		// Axis not coupled	
		IF NOT _stAXIS_REF.Status.Coupled THEN
			FB_MC2_AxisBasic_M_nMC_SetPositionRelative_iState:= 001;
		ELSE
			FB_MC2_AxisBasic_M_nMC_SetPositionRelative_iState:= 010;
		END_IF
	END_IF
ELSE
	FB_MC2_AxisBasic_M_nMC_SetPositionRelative_fbExecute_R_TRIG(CLK:= FALSE);
	FB_MC2_AxisBasic_M_nMC_SetPositionRelative_iState:= 000;
	IF FB_MC2_AxisBasic_M_nMC_SetPositionRelative_bExecute THEN
		M_nMC_SetPositionRelative:= Tc3_HBI_System.cMAPPING_ERROR;
	END_IF
	RETURN;
END_IF


//**********************************
// Main sequence
//**********************************
CASE FB_MC2_AxisBasic_M_nMC_SetPositionRelative_iState OF

	000: 	// Do nothing
	
	001:	// Set Axis position
			M_nMC_SetPositionRelative:= Tc3_HBI_System.cRUNNING;
			IF _stAXIS_REF.NcToPlc.AxisID > 0 THEN
				FB_MC2_AxisBasic_M_nMC_SetPositionRelative_fbMC2_SetPosition(Axis:= _stAXIS_REF, Execute:= FALSE); 
				FB_MC2_AxisBasic_M_nMC_SetPositionRelative_fbMC2_SetPosition(Axis:= _stAXIS_REF, Execute:= TRUE, Position:= FB_MC2_AxisBasic_M_nMC_SetPositionRelative_lrPosition); 
				FB_MC2_AxisBasic_M_nMC_SetPositionRelative_iState:= FB_MC2_AxisBasic_M_nMC_SetPositionRelative_iState +1;
			END_IF
			
	002:	// Set Axis position - Done
			M_nMC_SetPositionRelative:= Tc3_HBI_System.cRUNNING;
			FB_MC2_AxisBasic_M_nMC_SetPositionRelative_fbMC2_SetPosition(Axis:= _stAXIS_REF, Execute:= TRUE); 
			
			// Error handling
			IF FB_MC2_AxisBasic_M_nMC_SetPositionRelative_fbMC2_SetPosition.Error THEN
				M_nError(FB_MC2_AxisBasic_M_nMC_SetPositionRelative_fbMC2_SetPosition.ErrorID);
				M_nMC_SetPositionRelative:= FB_MC2_AxisBasic_M_nMC_SetPositionRelative_fbMC2_SetPosition.ErrorID;
			ELSE
				// Done
				IF FB_MC2_AxisBasic_M_nMC_SetPositionRelative_fbMC2_SetPosition.Done THEN
					FB_MC2_AxisBasic_M_nMC_SetPositionRelative_fbMC2_SetPosition(Axis:= _stAXIS_REF, Execute:= FALSE); 
					FB_MC2_AxisBasic_M_nMC_SetPositionRelative_iState:= 020;
				END_IF
			END_IF
		
	010:	// Coupled
			M_nMC_SetPositionRelative:= Tc3_HBI_System.cCOUPLED;
			IF NOT FB_MC2_AxisBasic_M_nMC_SetPositionRelative_bExecute THEN
				FB_MC2_AxisBasic_M_nMC_SetPositionRelative_fbMC2_SetPosition(Axis:= _stAXIS_REF, Execute:= FALSE); 
				FB_MC2_AxisBasic_M_nMC_SetPositionRelative_iState:= 000;
			END_IF	

	020:	// Done
			M_nMC_SetPositionRelative:= Tc3_HBI_System.cCOMPLETE;
			
			IF NOT FB_MC2_AxisBasic_M_nMC_SetPositionRelative_bExecute THEN
				FB_MC2_AxisBasic_M_nMC_SetPositionRelative_fbMC2_SetPosition(Axis:= _stAXIS_REF, Execute:= FALSE); 
				FB_MC2_AxisBasic_M_nMC_SetPositionRelative_iState:= 000;
			END_IF	
		
ELSE
	FB_MC2_AxisBasic_M_nMC_SetPositionRelative_iState:= 000;
END_CASE
END_METHOD

//	The result of the method is an unsigned double integer
//	0 = idle 
//	1 = coupled
//	2 = starting
//	3 = running
//	4 = aborted
// 	5 = no hardware connected
// 	6 = Spare
//	7 = pointer or index error
//	8 = mapping error
//	9 = parameter error
//	10 = complete
//	Any other number = ErrorID
METHOD PUBLIC M_nMC_SetScaleFactor : UDINT
VAR_INPUT
	bExecute: BOOL;
	lrScaleFactor: LREAL;
END_VAR
// Local variable
FB_MC2_AxisBasic_M_nMC_SetScaleFactor_bExecute:= bExecute;
FB_MC2_AxisBasic_M_nMC_SetScaleFactor_lrScaleFactor:= lrScaleFactor;

//**********************************
// Reset 
//**********************************
IF _bReset THEN
	IF _bError THEN
		FB_MC2_AxisBasic_M_nMC_SetScaleFactor_fbMC2_SetEncoderScalingFactor(Axis:= _stAXIS_REF, Execute:= FALSE);
		FB_MC2_AxisBasic_M_nMC_SetScaleFactor_iState:= 000;
	END_IF	
END_IF

//**********************************
// Wait for execute
//**********************************
IF _stAXIS_REF.NcToPlc.AxisID > 0 THEN
	FB_MC2_AxisBasic_M_nMC_SetScaleFactor_fbExecute_R_TRIG(CLK:= FB_MC2_AxisBasic_M_nMC_SetScaleFactor_bExecute);
	IF FB_MC2_AxisBasic_M_nMC_SetScaleFactor_fbExecute_R_TRIG.Q THEN
		FB_MC2_AxisBasic_M_nMC_SetScaleFactor_fbMC2_SetEncoderScalingFactor(Axis:= _stAXIS_REF, Execute:= FALSE, ScalingFactor:= FB_MC2_AxisBasic_M_nMC_SetScaleFactor_lrScaleFactor, Mode:= ENCODERSCALINGMODE_RELATIVE);
		
		// Axis not coupled	
		IF NOT _stAXIS_REF.Status.Coupled THEN
			FB_MC2_AxisBasic_M_nMC_SetScaleFactor_iState:= 001;
		ELSE
			FB_MC2_AxisBasic_M_nMC_SetScaleFactor_iState:= 010;
		END_IF
	END_IF
ELSE
	FB_MC2_AxisBasic_M_nMC_SetScaleFactor_fbExecute_R_TRIG(CLK:= FALSE);
	FB_MC2_AxisBasic_M_nMC_SetScaleFactor_iState:= 000;
	IF FB_MC2_AxisBasic_M_nMC_SetScaleFactor_bExecute THEN
		M_nMC_SetScaleFactor:= Tc3_HBI_System.cMAPPING_ERROR;
	END_IF
	RETURN;
END_IF

//**********************************
// Parameter check 
//**********************************
IF FB_MC2_AxisBasic_M_nMC_SetScaleFactor_bExecute THEN
	IF FB_MC2_AxisBasic_M_nMC_SetScaleFactor_lrScaleFactor = 0.0 THEN
		M_nMC_SetScaleFactor:= Tc3_HBI_System.cPARAMETER_ERROR;
		RETURN;
	END_IF
END_IF


//**********************************
// Main sequence
//**********************************
CASE FB_MC2_AxisBasic_M_nMC_SetScaleFactor_iState OF

	000: 	// Do nothing
	
	001:	// Check parameter input
			M_nMC_SetScaleFactor:= Tc3_HBI_System.cSTARTING;
			IF _stAXIS_REF.NcToPlc.AxisID > 0 THEN
				IF FB_MC2_AxisBasic_M_nMC_SetScaleFactor_lrScaleFactor > 0.0 THEN 
					FB_MC2_AxisBasic_M_nMC_SetScaleFactor_iState:= 2;
				ELSE
					M_nMC_SetScaleFactor:= Tc3_HBI_System.cPARAMETER_ERROR;
					IF NOT FB_MC2_AxisBasic_M_nMC_SetScaleFactor_bExecute THEN
						FB_MC2_AxisBasic_M_nMC_SetScaleFactor_iState:= 000;
					END_IF
				END_IF
			END_IF

	002:	// Set axis scale factor
			M_nMC_SetScaleFactor:= Tc3_HBI_System.cRUNNING;
			FB_MC2_AxisBasic_M_nMC_SetScaleFactor_fbMC2_SetEncoderScalingFactor(Axis:= _stAXIS_REF, Execute:= TRUE, ScalingFactor:= FB_MC2_AxisBasic_M_nMC_SetScaleFactor_lrScaleFactor, Mode:= ENCODERSCALINGMODE_RELATIVE);
			
			// Error handling
			IF FB_MC2_AxisBasic_M_nMC_SetScaleFactor_fbMC2_SetEncoderScalingFactor.Error THEN
				M_nError(FB_MC2_AxisBasic_M_nMC_SetScaleFactor_fbMC2_SetEncoderScalingFactor.ErrorID);
				M_nMC_SetScaleFactor:= FB_MC2_AxisBasic_M_nMC_SetScaleFactor_fbMC2_SetEncoderScalingFactor.ErrorID;
			ELSE
				// Done
				IF FB_MC2_AxisBasic_M_nMC_SetScaleFactor_fbMC2_SetEncoderScalingFactor.Done THEN
					FB_MC2_AxisBasic_M_nMC_SetScaleFactor_fbMC2_SetEncoderScalingFactor(Axis:= _stAXIS_REF, Execute:= FALSE);
					FB_MC2_AxisBasic_M_nMC_SetScaleFactor_iState:= 020;
				END_IF
			END_IF
		
	010:	// Coupled
			M_nMC_SetScaleFactor:= Tc3_HBI_System.cCOUPLED;
			IF NOT FB_MC2_AxisBasic_M_nMC_SetScaleFactor_bExecute THEN
				FB_MC2_AxisBasic_M_nMC_SetScaleFactor_fbMC2_SetEncoderScalingFactor(Axis:= _stAXIS_REF, Execute:= FALSE);
				FB_MC2_AxisBasic_M_nMC_SetScaleFactor_iState:= 000;
			END_IF	

	020:	// Done
			M_nMC_SetScaleFactor:= Tc3_HBI_System.cCOMPLETE;

			IF NOT FB_MC2_AxisBasic_M_nMC_SetScaleFactor_bExecute THEN
				FB_MC2_AxisBasic_M_nMC_SetScaleFactor_fbMC2_SetEncoderScalingFactor(Axis:= _stAXIS_REF, Execute:= FALSE);
				FB_MC2_AxisBasic_M_nMC_SetScaleFactor_iState:= 000;
			END_IF	

ELSE
	FB_MC2_AxisBasic_M_nMC_SetScaleFactor_iState:= 000;
END_CASE
END_METHOD

//	The result of the method is an unsigned double integer
//	0 = idle 
//	1 = coupled
//	2 = starting
//	3 = running
//	4 = aborted
// 	5 = no hardware connected
// 	6 = Spare
//	7 = pointer or index error
//	8 = mapping error
//	9 = parameter error
//	10 = complete
//	Any other number = ErrorID
METHOD PUBLIC M_nMC_SetVeloKvFactor : UDINT
VAR_INPUT
	bExecute: BOOL;
	lrKvFactor: LREAL;
END_VAR
// Local variable
FB_MC2_AxisBasic_M_nMC_SetVeloKvFactor_bExecute:= bExecute;
FB_MC2_AxisBasic_M_nMC_SetVeloKvFactor_lrKvFactor:= lrKvFactor;

//**********************************
// Reset 
//**********************************
IF _bReset THEN
	IF _bError THEN
		FB_MC2_AxisBasic_M_nMC_SetVeloKvFactor_fbADSWRITE(WRITE:= FALSE); 
		FB_MC2_AxisBasic_M_nMC_SetVeloKvFactor_iState:= 000;
	END_IF
END_IF

//**********************************
// Parameter check 
//**********************************
IF FB_MC2_AxisBasic_M_nMC_SetVeloKvFactor_bExecute THEN
	IF FB_MC2_AxisBasic_M_nMC_SetVeloKvFactor_lrKvFactor <= 0.0 THEN
		M_nMC_SetVeloKvFactor:= Tc3_HBI_System.cPARAMETER_ERROR;
		RETURN;
	END_IF	
END_IF


//**********************************
// Wait for execute
//**********************************
IF _stAXIS_REF.NcToPlc.AxisID > 0 THEN
	FB_MC2_AxisBasic_M_nMC_SetVeloKvFactor_fbExecute_R_TRIG(CLK:= FB_MC2_AxisBasic_M_nMC_SetVeloKvFactor_bExecute);
	IF FB_MC2_AxisBasic_M_nMC_SetVeloKvFactor_fbExecute_R_TRIG.Q THEN
		FB_MC2_AxisBasic_M_nMC_SetVeloKvFactor_iState:= 001;
	END_IF
ELSE
	FB_MC2_AxisBasic_M_nMC_SetVeloKvFactor_fbExecute_R_TRIG(CLK:= FALSE);
	FB_MC2_AxisBasic_M_nMC_SetVeloKvFactor_iState:= 000;
	IF FB_MC2_AxisBasic_M_nMC_SetVeloKvFactor_bExecute THEN
		M_nMC_SetVeloKvFactor:= Tc3_HBI_System.cMAPPING_ERROR;
	END_IF
	RETURN;
END_IF


//**********************************
// Main sequence
//**********************************
CASE FB_MC2_AxisBasic_M_nMC_SetVeloKvFactor_iState OF

	000: 	// Do nothing

	001:	// Set Velo Kv faktor
			IF FB_MC2_AxisBasic_M_nMC_SetVeloKvFactor_bExecute THEN				
				M_nMC_SetVeloKvFactor:= Tc3_HBI_System.cSTARTING;
				FB_MC2_AxisBasic_M_nMC_SetVeloKvFactor_fbADSWRITE(WRITE:= FALSE);
				FB_MC2_AxisBasic_M_nMC_SetVeloKvFactor_fbADSWRITE(
					NETID:= '', 
					PORT:= 501, 
					IDXGRP:= 16#6000 + _stAXIS_REF.NcToPlc.AxisId, 
					IDXOFFS:= 16#102, 
					LEN:= SIZEOF(FB_MC2_AxisBasic_M_nMC_SetVeloKvFactor_lrKvFactor), 
					SRCADDR:= ADR(FB_MC2_AxisBasic_M_nMC_SetVeloKvFactor_lrKvFactor), 
					WRITE:= TRUE, 
					TMOUT:= Tc2_System.DEFAULT_ADS_TIMEOUT, 
					BUSY=> , 
					ERR=> , 
					ERRID=> );
	 
				FB_MC2_AxisBasic_M_nMC_SetVeloKvFactor_iState:= FB_MC2_AxisBasic_M_nMC_SetVeloKvFactor_iState +1;
			ELSE
				FB_MC2_AxisBasic_M_nMC_SetVeloKvFactor_iState:= 000;
			END_IF	
	
	002:	// Done	
			M_nMC_SetVeloKvFactor:= Tc3_HBI_System.cRUNNING;	
			FB_MC2_AxisBasic_M_nMC_SetVeloKvFactor_fbADSWRITE(WRITE:= TRUE);
		
			// Error handling
			IF FB_MC2_AxisBasic_M_nMC_SetVeloKvFactor_fbADSWRITE.ERR THEN
				M_nError(nErrorID:= FB_MC2_AxisBasic_M_nMC_SetVeloKvFactor_fbADSWRITE.ERRID);
				M_nMC_SetVeloKvFactor:= FB_MC2_AxisBasic_M_nMC_SetVeloKvFactor_fbADSWRITE.ERRID;
			ELSE
				// Done
				IF NOT FB_MC2_AxisBasic_M_nMC_SetVeloKvFactor_fbADSWRITE.BUSY THEN
					FB_MC2_AxisBasic_M_nMC_SetVeloKvFactor_fbADSWRITE(WRITE:= FALSE); 
					FB_MC2_AxisBasic_M_nMC_SetVeloKvFactor_iState:= FB_MC2_AxisBasic_M_nMC_SetVeloKvFactor_iState +1;
				END_IF
			END_IF
			
	003:	// Done
			M_nMC_SetVeloKvFactor:= Tc3_HBI_System.cCOMPLETE;
			
			IF NOT FB_MC2_AxisBasic_M_nMC_SetVeloKvFactor_bExecute THEN	
				FB_MC2_AxisBasic_M_nMC_SetVeloKvFactor_iState:= 000;
			END_IF	
		
ELSE
	FB_MC2_AxisBasic_M_nMC_SetVeloKvFactor_iState:= 000;
END_CASE
END_METHOD

//	The result of the method is an unsigned double integer
//	0 = idle 
//	1 = coupled
//	2 = starting
//	3 = running
//	4 = aborted
// 	5 = no hardware connected
// 	6 = Spare
//	7 = pointer or index error
//	8 = mapping error
//	9 = parameter error
//	10 = complete
//	Any other number = ErrorID
METHOD PUBLIC M_nReset : UDINT
VAR_INPUT
	bExecute: BOOL;
END_VAR
// Local variable
FB_MC2_AxisBasic_M_nReset_bExecute:= bExecute;

//**********************************
// Wait for execute
//**********************************
FB_MC2_AxisBasic_M_nReset_fbExecute_R_TRIG(CLK:= FB_MC2_AxisBasic_M_nReset_bExecute);
IF FB_MC2_AxisBasic_M_nReset_fbExecute_R_TRIG.Q THEN
	FB_MC2_AxisBasic_M_nReset_fbMC2_Reset(Axis:= _stAXIS_REF, Execute:= FALSE);
	SUPER^.M_nReset(bExecute:= FALSE);
	FB_MC2_AxisBasic_M_nReset_bError:= _bError;
	FB_MC2_AxisBasic_M_nReset_iState:= 001;
END_IF	


//**********************************
// Main sequence
//**********************************
CASE FB_MC2_AxisBasic_M_nReset_iState OF

	000: 	// Do nothing
		
	001:	// Reset father	
			M_nReset:= Tc3_HBI_System.cRUNNING;
			FB_MC2_AxisBasic_M_nReset_nStatus:= SUPER^.M_nReset(bExecute:= TRUE);
			
			// Error handling
			IF FB_MC2_AxisBasic_M_nReset_nStatus > Tc3_HBI_System.cCOMPLETE THEN
				SUPER^.M_nReset(bExecute:= FALSE);		
				IF _stAXIS_REF.Status.Coupled THEN
					FB_MC2_AxisBasic_M_nReset_iState:= 020;
				ELSE
					FB_MC2_AxisBasic_M_nReset_iState:= 030;
				END_IF
			END_IF

			// Done
			IF FB_MC2_AxisBasic_M_nReset_nStatus = Tc3_HBI_System.cCOUPLED OR FB_MC2_AxisBasic_M_nReset_nStatus = Tc3_HBI_System.cCOMPLETE THEN
				SUPER^.M_nReset(bExecute:= FALSE);		
				IF _stAXIS_REF.Status.Coupled THEN
					FB_MC2_AxisBasic_M_nReset_iState:= 020;
				ELSE
					FB_MC2_AxisBasic_M_nReset_iState:= 030;
				END_IF
			END_IF
			
	020:	// Coupled
			M_nReset:= Tc3_HBI_System.cCOUPLED;
			IF NOT FB_MC2_AxisBasic_M_nReset_bExecute THEN
				FB_MC2_AxisBasic_M_nReset_fbMC2_Reset(Axis:= _stAXIS_REF, Execute:= FALSE);
				SUPER^.M_nReset(bExecute:= FALSE);		
				FB_MC2_AxisBasic_M_nReset_iState:= 000;
			END_IF	
	
	030:	// Done
			M_nReset:= Tc3_HBI_System.cCOMPLETE;
			IF NOT FB_MC2_AxisBasic_M_nReset_bExecute THEN
				FB_MC2_AxisBasic_M_nReset_fbMC2_Reset(Axis:= _stAXIS_REF, Execute:= FALSE);
				SUPER^.M_nReset(bExecute:= FALSE);		
				FB_MC2_AxisBasic_M_nReset_iState:= 000;
			END_IF

ELSE
	FB_MC2_AxisBasic_M_nReset_iState:= 000;
END_CASE
END_METHOD

PROPERTY PUBLIC P_bAdvancedSlaveDynamics : BOOL
SET
FB_MC2_AxisBasic_M_nMC_GearInMultiMaster_bAdvancedSlaveDynamics:= P_bAdvancedSlaveDynamics;
END_SET
END_PROPERTY

PROPERTY PUBLIC P_bInGear : BOOL
GET
P_bInGear:= _stAXIS_REF.Status.Coupled;
END_GET
END_PROPERTY

PROPERTY PUBLIC P_lrAbsolutePhaseShift  : lreal
GET
P_lrAbsolutePhaseShift:= FB_MC2_AxisBasic_M_nMC_PhasingAbsolute_lrAbsolutePhaseShift;
END_GET
END_PROPERTY

PROPERTY PUBLIC P_lrCoveredPhaseShift : lreal
GET
P_lrCoveredPhaseShift:= FB_MC2_AxisBasic_M_nMC_PhasingRelative_lrCoveredPhaseShift;
END_GET
END_PROPERTY

PROPERTY PUBLIC P_lrGearRatio1 : LREAL
SET
FB_MC2_AxisBasic_M_nMC_GearInMultiMaster_lrGearRatio1:= P_lrGearRatio1;
END_SET
END_PROPERTY

PROPERTY PUBLIC P_lrGearRatio2 : LREAL
SET
FB_MC2_AxisBasic_M_nMC_GearInMultiMaster_lrGearRatio2:= P_lrGearRatio2;
END_SET
END_PROPERTY

PROPERTY PUBLIC P_lrGearRatio3 : LREAL
SET
FB_MC2_AxisBasic_M_nMC_GearInMultiMaster_lrGearRatio3:= P_lrGearRatio3;
END_SET
END_PROPERTY

PROPERTY PUBLIC P_lrGearRatio4 : LREAL
SET
FB_MC2_AxisBasic_M_nMC_GearInMultiMaster_lrGearRatio4:= P_lrGearRatio4;
END_SET
END_PROPERTY

PROPERTY PUBLIC P_lrMaxVelocity : LREAL
GET
P_lrMaxVelocity:= FB_MC2_AxisBasic_M_nMC_ReadParameter_lrMaxVelocity;
END_GET
END_PROPERTY

PROPERTY PUBLIC P_lrModuloFactor : LREAL
GET
IF FB_MC2_AxisBasic_M_nMC_SetModuloFactor_lrModuloFactor = 0 THEN
	FB_MC2_AxisBasic_M_nMC_SetModuloFactor_lrModuloFactor:= 360.0;
	P_lrModuloFactor:= FB_MC2_AxisBasic_M_nMC_SetModuloFactor_lrModuloFactor;
ELSE
	P_lrModuloFactor:= FB_MC2_AxisBasic_M_nMC_SetModuloFactor_lrModuloFactor;
END_IF
END_GET
END_PROPERTY

END_FUNCTION_BLOCK

// MOTION/POUs/FBs/Compact/FB_MC2_Compact
//------------------------------------------------------------------------------------------
//                                                                                        	
//***************************** Beckhoff TwinCAT Examples **********************************
//                                                                                        	
//************************************* WARNING ********************************************
// This program is only an example. If it is used as a control program in any real        	
// application, Beckhoff is not responsible for any malfunction, loss or damage           	
// which could arise by using this program!                                               	
//                                                                                        	
//*************************************  Program Info. *************************************
//                                                                                        	
// PLC program name:       	FB_MC2_Compact (FB)                                          	
// Hardware platform:      	TwinCat PTP v3.1.4022				                          	                                  	
//                                                                                        	
// ======================================================================================== 
//         Version       Date                        Remarks                              	
// ======================================================================================== 
//         3.1      27 feb 2018                First release of this example  
//         3.7.1.1		 09 may 2018    			 Next release of this example   
// ======================================================================================== 
//                                                                                        	
//******************************* Aims OF this PLC PROGRAM *********************************
//                                                                                        	
// MC2 servo axis compact						 			                                      	
// Add axis error message 																                      	
//                                                                                        	
//----------------------------------------------------------------------------------------- 
FUNCTION_BLOCK FB_MC2_Compact EXTENDS FB_Basic IMPLEMENTS I_MC2_Compact
VAR
//***************************
// Property variables
//***************************
	_stAXIS_REF: Tc2_MC2.AXIS_REF;
	_eBufferMode: MC_BufferMode:= Tc2_MC2.MC_Aborting;
	_bHardwareConnected: BOOL;	
	_stDriveAddress: ST_DriveAddress;
	_stDynamic: _ST_MC2_Dynamic;
	_sMessage: STRING(80);
	
//***************************
// Metods variable
//***************************
	FB_MC2_Compact_M_nMC_Dynamic_bExecute: BOOL;
	FB_MC2_Compact_M_nMC_Dynamic_lrAcceleration: LREAL;
	FB_MC2_Compact_M_nMC_Dynamic_lrDeceleration: LREAL;
	FB_MC2_Compact_M_nMC_Dynamic_lrJerk: LREAL;

	FB_MC2_Compact_M_nMC_Halt_bExecute: BOOL;
	FB_MC2_Compact_M_nMC_Halt_iState: INT;
	FB_MC2_Compact_M_nMC_Halt_fbExecute_R_TRIG: R_TRIG;
	FB_MC2_Compact_M_nMC_Halt_fbMC2_Halt1: Tc2_MC2.MC_Halt;
	FB_MC2_Compact_M_nMC_Halt_fbMC2_Halt2: Tc2_MC2.MC_Halt;

	FB_MC2_Compact_M_nMC_Home_bExecute: BOOL;
	FB_MC2_Compact_M_nMC_Home_lrPosition: LREAL;
	FB_MC2_Compact_M_nMC_Home_bCalibrationCam: BOOL;
	FB_MC2_Compact_M_nMC_Home_eHomingMode: MC_HomingMode;
	FB_MC2_Compact_M_nMC_Home_iState: INT;
	FB_MC2_Compact_M_nMC_Home_fbExecute_R_TRIG: Tc2_Standard.R_TRIG;
	FB_MC2_Compact_M_nMC_Home_fbMC2_Halt: Tc2_MC2.MC_Halt;
	FB_MC2_Compact_M_nMC_Home_fbMC2_Home: Tc2_MC2.MC_Home;
	
	FB_MC2_Compact_M_nMC_HomeReset_bExecute: BOOL;
	FB_MC2_Compact_M_nMC_HomeReset_iState: INT;
	FB_MC2_Compact_M_nMC_HomeReset_fbExecute_R_TRIG: Tc2_Standard.R_TRIG;
	FB_MC2_Compact_M_nMC_HomeReset_fbMC2_Home: Tc2_MC2.MC_Home;

	FB_MC2_Compact_M_nMC_Jog_bForward: BOOL;
	FB_MC2_Compact_M_nMC_Jog_bBackwards: BOOL;
	FB_MC2_Compact_M_nMC_Jog_lrVelocity: LREAL;
	FB_MC2_Compact_M_nMC_Jog_iState: INT;
	FB_MC2_Compact_M_nMC_Jog_fbExecute_R_TRIG1: R_TRIG;
	FB_MC2_Compact_M_nMC_Jog_fbExecute_R_TRIG2: R_TRIG;
	FB_MC2_Compact_M_nMC_Jog_fbMC2_Jog1: Tc2_MC2.MC_Jog;
	FB_MC2_Compact_M_nMC_Jog_fbMC2_Jog2: Tc2_MC2.MC_Jog;

	FB_MC2_Compact_M_nMC_Local_Halt_bExecute: BOOL;
	FB_MC2_Compact_M_nMC_Local_Halt_iState: INT;
	FB_MC2_Compact_M_nMC_Local_Halt_fbExecute_R_TRIG: R_TRIG;
	FB_MC2_Compact_M_nMC_Local_Halt_fbMC2_Halt1: Tc2_MC2.MC_Halt;
	FB_MC2_Compact_M_nMC_Local_Halt_fbMC2_Halt2: Tc2_MC2.MC_Halt;

	FB_MC2_Compact_M_nMC_MoveAbsolute_bExecute: BOOL;
	FB_MC2_Compact_M_nMC_MoveAbsolute_lrPosition: LREAL;
	FB_MC2_Compact_M_nMC_MoveAbsolute_lrVelocity: LREAL;
	FB_MC2_Compact_M_nMC_MoveAbsolute_iState: INT;
	FB_MC2_Compact_M_nMC_MoveAbsolute_fbExecute_R_TRIG: Tc2_Standard.R_TRIG;
	FB_MC2_Compact_M_nMC_MoveAbsolute_fbMC2_MoveAbsolute1: Tc2_MC2.MC_MoveAbsolute;
	FB_MC2_Compact_M_nMC_MoveAbsolute_fbMC2_MoveAbsolute2: Tc2_MC2.MC_MoveAbsolute;

	FB_MC2_Compact_M_nMC_MoveModulo_bExecute: BOOL;
	FB_MC2_Compact_M_nMC_MoveModulo_lrPosition: LREAL;
	FB_MC2_Compact_M_nMC_MoveModulo_lrVelocity: LREAL;
	FB_MC2_Compact_M_nMC_MoveModulo_eDirection: Tc2_MC2.MC_Direction;
	FB_MC2_Compact_M_nMC_MoveModulo_iState: INT;
	FB_MC2_Compact_M_nMC_MoveModulo_fbExecute_R_TRIG: Tc2_Standard.R_TRIG;
	FB_MC2_Compact_M_nMC_MoveModulo_fbMC2_MoveModulo1: Tc2_MC2.MC_MoveModulo;
	FB_MC2_Compact_M_nMC_MoveModulo_fbMC2_MoveModulo2: Tc2_MC2.MC_MoveModulo;

	FB_MC2_Compact_M_nMC_MoveRelative_bExecute: BOOL;
	FB_MC2_Compact_M_nMC_MoveRelative_lrDistance: LREAL;
	FB_MC2_Compact_M_nMC_MoveRelative_lrVelocity: LREAL;
	FB_MC2_Compact_M_nMC_MoveRelative_iState: INT;
	FB_MC2_Compact_M_nMC_MoveRelative_fbExecute_R_TRIG: Tc2_Standard.R_TRIG;
	FB_MC2_Compact_M_nMC_MoveRelative_fbMC2_MoveRelative1: Tc2_MC2.MC_MoveRelative;
	FB_MC2_Compact_M_nMC_MoveRelative_fbMC2_MoveRelative2: Tc2_MC2.MC_MoveRelative;

	FB_MC2_Compact_M_nMC_MoveVelocity_bExecute: BOOL;
	FB_MC2_Compact_M_nMC_MoveVelocity_lrVelocity: LREAL;
	FB_MC2_Compact_M_nMC_MoveVelocity_eDirection: MC_Direction;
	FB_MC2_Compact_M_nMC_MoveVelocity_iState: INT;
	FB_MC2_Compact_M_nMC_MoveVelocity_fbExecute_R_TRIG: Tc2_Standard.R_TRIG;
	FB_MC2_Compact_M_nMC_MoveVelocity_fbMC2_MoveVelocity1: Tc2_MC2.MC_MoveVelocity;
	FB_MC2_Compact_M_nMC_MoveVelocity_fbMC2_MoveVelocity2: Tc2_MC2.MC_MoveVelocity;
	
	FB_MC2_Compact_M_nMC_Power_bEnable: BOOL;
	FB_MC2_Compact_M_nMC_Power_bE_Stop: BOOL;
	FB_MC2_Compact_M_nMC_Power_bE_StopDelay: BOOL;
	FB_MC2_Compact_M_nMC_Power_bEnable_Positive: BOOL;
	FB_MC2_Compact_M_nMC_Power_bEnable_Negative: BOOL;
	FB_MC2_Compact_M_nMC_Power_lrOverride: LREAL := 100.0;
	FB_MC2_Compact_M_nMC_Power_fbStartDelay_TON: Tc2_Standard.TON;
	FB_MC2_Compact_M_nMC_Power_arr_fb_R_TRIG: ARRAY[1..12] OF Tc2_Standard.R_TRIG;
	FB_MC2_Compact_M_nMC_Power_arr_nRet: ARRAY[1..4] OF UDINT;
	FB_MC2_Compact_M_nMC_Power_fbMC2_Power: Tc2_MC2.MC_Power;
	FB_MC2_Compact_M_nMC_Power_fbDelay_TON: Tc2_Standard.TON;
	FB_MC2_Compact_M_nMC_Power_fbPuls_TON: Tc2_Standard.TON;
	FB_MC2_Compact_M_nMC_Power_bReset: BOOL;
	FB_MC2_Compact_M_nMC_Power_iResetState: INT;
	FB_MC2_Compact_M_nMC_Power_bLocal_Halt: BOOL;
	FB_MC2_Compact_M_nMC_Power_bError: BOOL;
	
	FB_MC2_Compact_M_nMC_QuickStop_bExecute: BOOL;
	FB_MC2_Compact_M_nMC_QuickStop_lrDeceleration: LREAL;
	FB_MC2_Compact_M_nMC_QuickStop_lrJerk: LREAL;
	FB_MC2_Compact_M_nMC_QuickStop_bQuickStopRunning: BOOL;
	FB_MC2_Compact_M_nMC_QuickStop_iState: INT;
	FB_MC2_Compact_M_nMC_QuickStop_fbExecute_R_TRIG: Tc2_Standard.R_TRIG;
	FB_MC2_Compact_M_nMC_QuickStop_fbMC2_Stop: Tc2_MC2.MC_Stop;

	FB_MC2_Compact_M_nMC_ReadDriveAddress_bExecute: BOOL;
	FB_MC2_Compact_M_nMC_ReadDriveAddress_iState: INT;
	FB_MC2_Compact_M_nMC_ReadDriveAddress_bError: BOOL;
	FB_MC2_Compact_M_nMC_ReadDriveAddress_fbReadDriveAddress: Tc2_MC2.MC_ReadDriveAddress;

	FB_MC2_Compact_M_nMC_Stop_bExecute: BOOL;
	FB_MC2_Compact_M_nMC_Stop_iState: INT;
	FB_MC2_Compact_M_nMC_Stop_fbExecute_R_TRIG: R_TRIG;
	FB_MC2_Compact_M_nMC_Stop_fbMC2_Stop1: Tc2_MC2.MC_Stop;
	FB_MC2_Compact_M_nMC_Stop_fbMC2_Stop2: Tc2_MC2.MC_Stop;

	FB_MC2_Compact_M_nReset_bExecute: BOOL;
	FB_MC2_Compact_M_nReset_iState: INT;
	FB_MC2_Compact_M_nReset_fbExecute_R_TRIG: Tc2_Standard.R_TRIG;
	FB_MC2_Compact_M_nReset_fbMC2_Reset: Tc2_MC2.MC_Reset;
	FB_MC2_Compact_M_nReset_fbMC2_Stop: Tc2_MC2.MC_Stop;
	FB_MC2_Compact_M_nReset_nStatus: UDINT;
END_VAR

//	The result of the method is an unsigned double integer
//	0 = idle 
//	1 = coupled
//	2 = starting
//	3 = running
//	4 = aborted
// 	5 = no hardware connected
// 	6 = Spare
//	7 = pointer or index error
//	8 = mapping error
//	9 = parameter error
//	10 = complete
//	Any other number = ErrorID
METHOD PUBLIC M_nMC_Dynamic : UDINT
VAR_INPUT
	bExecute: BOOL;
	lrAcceleration: LREAL;
	lrDeceleration: LREAL;
	lrJerk: LREAL;
END_VAR
// Local variable
FB_MC2_Compact_M_nMC_Dynamic_bExecute:= bExecute;
FB_MC2_Compact_M_nMC_Dynamic_lrAcceleration:= lrAcceleration;
FB_MC2_Compact_M_nMC_Dynamic_lrDeceleration:= lrDeceleration;
FB_MC2_Compact_M_nMC_Dynamic_lrJerk:= lrJerk;

//**********************************
// Parameter check 
//**********************************
IF FB_MC2_Compact_M_nMC_Dynamic_bExecute THEN
	IF FB_MC2_Compact_M_nMC_Dynamic_lrAcceleration < 0.0 OR FB_MC2_Compact_M_nMC_Dynamic_lrDeceleration < 0.0 OR FB_MC2_Compact_M_nMC_Dynamic_lrJerk < 0.0 THEN
		M_nMC_Dynamic:= Tc3_HBI_System.cPARAMETER_ERROR;
		RETURN;
	END_IF

	// Check for Axis
	IF _stAXIS_REF.NcToPlc.AxisID = 0 THEN
		RETURN;
	ELSE	
		// Update dynamic
		THIS^._stDynamic.lrAcceleration:= FB_MC2_Compact_M_nMC_Dynamic_lrAcceleration;
		THIS^._stDynamic.lrDeceleration:= FB_MC2_Compact_M_nMC_Dynamic_lrDeceleration;
		THIS^._stDynamic.lrJerk:= FB_MC2_Compact_M_nMC_Dynamic_lrJerk;
		M_nMC_Dynamic:= Tc3_HBI_System.cCOMPLETE;
	END_IF
	
END_IF
END_METHOD

//	The result of the method is an unsigned double integer
//	0 = idle 
//	1 = coupled
//	2 = starting
//	3 = running
//	4 = aborted
// 	5 = no hardware connected
// 	6 = Spare
//	7 = pointer or index error
//	8 = mapping error
//	9 = parameter error
//	10 = complete
//	Any other number = ErrorID
METHOD PUBLIC M_nMC_Halt : UDINT
VAR_INPUT
	bExecute: BOOL;
END_VAR
// Local variable
FB_MC2_Compact_M_nMC_Halt_bExecute:= bExecute;

//**********************************
// Reset 
//**********************************
IF _bReset THEN
	IF _bError THEN
		FB_MC2_Compact_M_nMC_Halt_fbMC2_Halt1(Axis:= _stAXIS_REF, Execute:= FALSE);
		FB_MC2_Compact_M_nMC_Halt_fbMC2_Halt2(Axis:= _stAXIS_REF, Execute:= FALSE);
		FB_MC2_Compact_M_nMC_Halt_iState:= 000;
		_sMessage:= '';
	END_IF
END_IF

//**********************************
// Wait for execute
//**********************************
IF _stAXIS_REF.NcToPlc.AxisID > 0 THEN
	FB_MC2_Compact_M_nMC_Halt_fbExecute_R_TRIG(CLK:= FB_MC2_Compact_M_nMC_Halt_bExecute);
	IF FB_MC2_Compact_M_nMC_Halt_fbExecute_R_TRIG.Q THEN
			FB_MC2_Compact_M_nMC_Halt_fbMC2_Halt1(Axis:= _stAXIS_REF, Deceleration:= _stDynamic.lrDeceleration, Jerk:= _stDynamic.lrJerk, BufferMode:= _eBufferMode);
			FB_MC2_Compact_M_nMC_Halt_fbMC2_Halt2(Axis:= _stAXIS_REF, Deceleration:= _stDynamic.lrDeceleration, Jerk:= _stDynamic.lrJerk, BufferMode:= _eBufferMode);
	
			// Axis not coupled	
			IF NOT _stAXIS_REF.Status.Coupled THEN
				IF FB_MC2_Compact_M_nMC_Halt_fbMC2_Halt1.Execute OR FB_MC2_Compact_M_nMC_Halt_fbMC2_Halt1.Busy THEN
					FB_MC2_Compact_M_nMC_Halt_fbMC2_Halt1(Axis:= _stAXIS_REF, Execute:= FALSE);
					FB_MC2_Compact_M_nMC_Halt_fbMC2_Halt2(Axis:= _stAXIS_REF, Execute:= FALSE);
					FB_MC2_Compact_M_nMC_Halt_fbMC2_Halt2.Execute:= TRUE;
					FB_MC2_Compact_M_nMC_Halt_iState:= 010;
				ELSE
					FB_MC2_Compact_M_nMC_Halt_fbMC2_Halt1(Axis:= _stAXIS_REF, Execute:= FALSE);
					FB_MC2_Compact_M_nMC_Halt_fbMC2_Halt2(Axis:= _stAXIS_REF, Execute:= FALSE);
					FB_MC2_Compact_M_nMC_Halt_fbMC2_Halt1.Execute:= TRUE;
					FB_MC2_Compact_M_nMC_Halt_iState:= 001;
				END_IF
			ELSE
				FB_MC2_Compact_M_nMC_Halt_fbMC2_Halt1(Axis:= _stAXIS_REF, Execute:= FALSE);
				FB_MC2_Compact_M_nMC_Halt_fbMC2_Halt2(Axis:= _stAXIS_REF, Execute:= FALSE);
				FB_MC2_Compact_M_nMC_Halt_iState:= 030;
			END_IF
		
	END_IF
ELSE
	FB_MC2_Compact_M_nMC_Halt_fbExecute_R_TRIG(CLK:= FALSE);
	FB_MC2_Compact_M_nMC_Halt_iState:= 000;
	IF bExecute THEN
		M_nMC_Halt:= Tc3_HBI_System.cMAPPING_ERROR;
	END_IF
	RETURN;
END_IF


//**********************************
// Main sequence
//**********************************
CASE FB_MC2_Compact_M_nMC_Halt_iState OF

	000: 	// Do nothing
	
	001:	// Stop Axis1
			M_nMC_Halt:= Tc3_HBI_System.cSTARTING;
			FB_MC2_Compact_M_nMC_Halt_fbMC2_Halt1(Axis:= _stAXIS_REF);
			FB_MC2_Compact_M_nMC_Halt_fbMC2_Halt2(Axis:= _stAXIS_REF);
		
			// Command aborted
			IF FB_MC2_Compact_M_nMC_Halt_fbMC2_Halt1.CommandAborted THEN
				FB_MC2_Compact_M_nMC_Halt_fbMC2_Halt2.Execute:= FALSE;
				FB_MC2_Compact_M_nMC_Halt_iState:= 040;
			ELSE
				// Error handling
				IF FB_MC2_Compact_M_nMC_Halt_fbMC2_Halt1.Error THEN
					M_nError(FB_MC2_Compact_M_nMC_Halt_fbMC2_Halt1.ErrorID);
					M_nMC_Halt:= FB_MC2_Compact_M_nMC_Halt_fbMC2_Halt1.ErrorID;
					_sMessage:= 'Axis Halt Error';
				ELSE
					// Active
					IF FB_MC2_Compact_M_nMC_Halt_fbMC2_Halt1.Active THEN
						FB_MC2_Compact_M_nMC_Halt_iState:= 002;
					ELSE
						// Done
						IF FB_MC2_Compact_M_nMC_Halt_fbMC2_Halt1.Done THEN
							FB_MC2_Compact_M_nMC_Halt_iState:= 040;
						END_IF
					END_IF	
				END_IF
			END_IF
	
	002:	// Stop Axis
			M_nMC_Halt:= Tc3_HBI_System.cRUNNING;
			FB_MC2_Compact_M_nMC_Halt_fbMC2_Halt1(Axis:= _stAXIS_REF);
			FB_MC2_Compact_M_nMC_Halt_fbMC2_Halt2(Axis:= _stAXIS_REF);
	
			// Command aborted
			IF FB_MC2_Compact_M_nMC_Halt_fbMC2_Halt1.CommandAborted THEN
				FB_MC2_Compact_M_nMC_Halt_fbMC2_Halt2.Execute:= FALSE;
				FB_MC2_Compact_M_nMC_Halt_iState:= 040;
			ELSE
				// Error handling
				IF FB_MC2_Compact_M_nMC_Halt_fbMC2_Halt1.Error THEN
					M_nError(FB_MC2_Compact_M_nMC_Halt_fbMC2_Halt1.ErrorID);
					M_nMC_Halt:= FB_MC2_Compact_M_nMC_Halt_fbMC2_Halt1.ErrorID;
					_sMessage:= 'Axis Halt Error';
				ELSE
					// Done
					IF FB_MC2_Compact_M_nMC_Halt_fbMC2_Halt1.Done THEN
						FB_MC2_Compact_M_nMC_Halt_iState:= 040;
					END_IF
				END_IF
			END_IF 
	
	010:	// Stop Axis1
			M_nMC_Halt:= Tc3_HBI_System.cSTARTING;
			FB_MC2_Compact_M_nMC_Halt_fbMC2_Halt1(Axis:= _stAXIS_REF);
			FB_MC2_Compact_M_nMC_Halt_fbMC2_Halt2(Axis:= _stAXIS_REF);
			
			// Command aborted
			IF FB_MC2_Compact_M_nMC_Halt_fbMC2_Halt2.CommandAborted THEN
				FB_MC2_Compact_M_nMC_Halt_fbMC2_Halt1.Execute:= FALSE;
				FB_MC2_Compact_M_nMC_Halt_iState:= 040;
			ELSE
				// Error handling
				IF FB_MC2_Compact_M_nMC_Halt_fbMC2_Halt2.Error THEN
					M_nError(FB_MC2_Compact_M_nMC_Halt_fbMC2_Halt2.ErrorID);
					M_nMC_Halt:= FB_MC2_Compact_M_nMC_Halt_fbMC2_Halt2.ErrorID;
					_sMessage:= 'Axis Halt Error';
				ELSE
					// Active
					IF FB_MC2_Compact_M_nMC_Halt_fbMC2_Halt2.Active THEN
						FB_MC2_Compact_M_nMC_Halt_iState:= 011;
					ELSE
						// Done
						IF FB_MC2_Compact_M_nMC_Halt_fbMC2_Halt2.Done THEN
							FB_MC2_Compact_M_nMC_Halt_iState:= 040;
						END_IF
					END_IF	
				END_IF
			END_IF 
		
	011:	// Stop Axis2
			M_nMC_Halt:= Tc3_HBI_System.cRUNNING;
			FB_MC2_Compact_M_nMC_Halt_fbMC2_Halt1(Axis:= _stAXIS_REF);
			FB_MC2_Compact_M_nMC_Halt_fbMC2_Halt2(Axis:= _stAXIS_REF);
			
			// Command aborted
			IF FB_MC2_Compact_M_nMC_Halt_fbMC2_Halt2.CommandAborted THEN
				FB_MC2_Compact_M_nMC_Halt_fbMC2_Halt1.Execute:= FALSE;
				FB_MC2_Compact_M_nMC_Halt_iState:= 040;
			ELSE
				// Error handling
				IF FB_MC2_Compact_M_nMC_Halt_fbMC2_Halt2.Error THEN
					M_nError(FB_MC2_Compact_M_nMC_Halt_fbMC2_Halt2.ErrorID);
					M_nMC_Halt:= FB_MC2_Compact_M_nMC_Halt_fbMC2_Halt2.ErrorID;
					_sMessage:= 'Axis Halt Error';
				ELSE
					// Done
					IF FB_MC2_Compact_M_nMC_Halt_fbMC2_Halt2.Done THEN
						FB_MC2_Compact_M_nMC_Halt_iState:= 040;
					END_IF
				END_IF
			END_IF
	
	030:	// Coupled
			M_nMC_Halt:= Tc3_HBI_System.cCOUPLED;
			FB_MC2_Compact_M_nMC_Halt_fbMC2_Halt1(Axis:= _stAXIS_REF);
			FB_MC2_Compact_M_nMC_Halt_fbMC2_Halt2(Axis:= _stAXIS_REF);

			IF NOT FB_MC2_Compact_M_nMC_Halt_bExecute THEN
				FB_MC2_Compact_M_nMC_Halt_fbMC2_Halt1(Axis:= _stAXIS_REF, Execute:= FALSE);
				FB_MC2_Compact_M_nMC_Halt_fbMC2_Halt2(Axis:= _stAXIS_REF, Execute:= FALSE);
				FB_MC2_Compact_M_nMC_Halt_iState:= 000;
			END_IF	

	040:	// Done
			M_nMC_Halt:= Tc3_HBI_System.cCOMPLETE;
			FB_MC2_Compact_M_nMC_Halt_fbMC2_Halt1(Axis:= _stAXIS_REF);
			FB_MC2_Compact_M_nMC_Halt_fbMC2_Halt2(Axis:= _stAXIS_REF);
			
			IF FB_MC2_Compact_M_nMC_Halt_bExecute THEN
				IF FB_MC2_Compact_M_nMC_Halt_fbMC2_Halt1.Execute AND FB_MC2_Compact_M_nMC_Halt_fbMC2_Halt1.CommandAborted THEN
					M_nMC_Halt:= Tc3_HBI_System.cABORTED;
				END_IF
				IF FB_MC2_Compact_M_nMC_Halt_fbMC2_Halt2.Execute AND FB_MC2_Compact_M_nMC_Halt_fbMC2_Halt2.CommandAborted THEN
					M_nMC_Halt:= Tc3_HBI_System.cABORTED;
				END_IF
			ELSE
				FB_MC2_Compact_M_nMC_Halt_fbMC2_Halt1(Axis:= _stAXIS_REF, Execute:= FALSE);
				FB_MC2_Compact_M_nMC_Halt_fbMC2_Halt2(Axis:= _stAXIS_REF, Execute:= FALSE);
				FB_MC2_Compact_M_nMC_Halt_iState:= 000;
			END_IF	
		
ELSE
	FB_MC2_Compact_M_nMC_Halt_iState:= 000;
END_CASE
END_METHOD

//	The result of the method is an unsigned double integer
//	0 = idle 
//	1 = coupled
//	2 = starting
//	3 = running
//	4 = aborted
// 	5 = no hardware connected
// 	6 = Spare
//	7 = pointer or index error
//	8 = mapping error
//	9 = parameter error
//	10 = complete
//	Any other number = ErrorID
METHOD PUBLIC M_nMC_Home : UDINT
VAR_INPUT
	bExecute: BOOL;
	lrPosition: LREAL;
	bCalibrationCam: BOOL;
	eHomingMode: MC_HomingMode;
END_VAR
// Local variable
FB_MC2_Compact_M_nMC_Home_bExecute:= bExecute;
FB_MC2_Compact_M_nMC_Home_lrPosition:= lrPosition;
FB_MC2_Compact_M_nMC_Home_bCalibrationCam:= bCalibrationCam;
FB_MC2_Compact_M_nMC_Home_eHomingMode:= eHomingMode; 

//**********************************
// Reset 
//**********************************
IF _bReset THEN
	IF _bError THEN
		FB_MC2_Compact_M_nMC_Home_fbMC2_Halt(Axis:= _stAXIS_REF, Execute:= FALSE); 
		FB_MC2_Compact_M_nMC_Home_fbMC2_Home(Axis:= _stAXIS_REF, Execute:= FALSE);
		FB_MC2_Compact_M_nMC_Home_iState:= 000;
		_sMessage:= '';
	END_IF
END_IF

//**********************************
// Wait for execute
//**********************************
IF _stAXIS_REF.NcToPlc.AxisID > 0 THEN
	FB_MC2_Compact_M_nMC_Home_fbExecute_R_TRIG(CLK:= FB_MC2_Compact_M_nMC_Home_bExecute);
	IF FB_MC2_Compact_M_nMC_Home_fbExecute_R_TRIG.Q THEN
		FB_MC2_Compact_M_nMC_Home_fbMC2_Halt(Axis:= _stAXIS_REF, Execute:= FALSE, Deceleration:= _stDynamic.lrDeceleration, Jerk:= _stDynamic.lrJerk);
		FB_MC2_Compact_M_nMC_Home_fbMC2_Home(Axis:= _stAXIS_REF, Execute:= FALSE, Position:= FB_MC2_Compact_M_nMC_Home_lrPosition, HomingMode:= FB_MC2_Compact_M_nMC_Home_eHomingMode, BufferMode:= MC_Aborting, bCalibrationCam:= FB_MC2_Compact_M_nMC_Home_bCalibrationCam);	
	
		// Axis not coupled	
		IF NOT _stAXIS_REF.Status.Coupled THEN
			FB_MC2_Compact_M_nMC_Home_iState:= 001;
		ELSE
			FB_MC2_Compact_M_nMC_Home_iState:= 020;
		END_IF
		
	END_IF
ELSE
	FB_MC2_Compact_M_nMC_Home_fbExecute_R_TRIG(CLK:= FALSE);
	FB_MC2_Compact_M_nMC_Home_iState:= 000;
	IF FB_MC2_Compact_M_nMC_Home_bExecute THEN
		M_nMC_Home:= Tc3_HBI_System.cMAPPING_ERROR;
	END_IF
	RETURN;
END_IF


//**********************************
// Main sequence
//**********************************
CASE FB_MC2_Compact_M_nMC_Home_iState OF

	000: 	// Do nothing
	
	001:	// Stop Axis
			M_nMC_Home:= Tc3_HBI_System.cSTARTING;
			FB_MC2_Compact_M_nMC_Home_fbMC2_Halt(Axis:= _stAXIS_REF, Execute:= TRUE, Deceleration:= _stDynamic.lrDeceleration, Jerk:= _stDynamic.lrJerk);
	
			// Command aborted
			IF FB_MC2_Compact_M_nMC_Home_fbMC2_Halt.CommandAborted THEN
				FB_MC2_Compact_M_nMC_Home_iState:= 030;
			ELSE
				// Error handling
				IF FB_MC2_Compact_M_nMC_Home_fbMC2_Halt.Error THEN
					M_nError(nErrorID:= FB_MC2_Compact_M_nMC_Home_fbMC2_Halt.ErrorID);
					M_nMC_Home:= FB_MC2_Compact_M_nMC_Home_fbMC2_Halt.ErrorID;
					_sMessage:= 'Axis Home Error';
				ELSE
					// Done
					IF FB_MC2_Compact_M_nMC_Home_fbMC2_Halt.Done THEN
						FB_MC2_Compact_M_nMC_Home_iState:= 010;
					END_IF	
				END_IF
			END_IF
		
	010:	// Home axis
			FB_MC2_Compact_M_nMC_Home_fbMC2_Home(Axis:= _stAXIS_REF, Execute:= TRUE, Position:= FB_MC2_Compact_M_nMC_Home_lrPosition, HomingMode:= FB_MC2_Compact_M_nMC_Home_eHomingMode, BufferMode:= MC_Aborting, bCalibrationCam:= FB_MC2_Compact_M_nMC_Home_bCalibrationCam);	
		
			IF eHomingMode = MC_DefaultHoming THEN
				IF _stAXIS_REF.Status.Moving THEN
					M_nMC_Home:= Tc3_HBI_System.cRUNNING;
				ELSE
					M_nMC_Home:= Tc3_HBI_System.cSTARTING;
				END_IF
			ELSE
				IF FB_MC2_Compact_M_nMC_Home_fbMC2_Home.Busy THEN
					M_nMC_Home:= Tc3_HBI_System.cRUNNING;
				ELSE
					M_nMC_Home:= Tc3_HBI_System.cSTARTING;
				END_IF
			END_IF
			
			// Command aborted
			IF FB_MC2_Compact_M_nMC_Home_fbMC2_Home.CommandAborted THEN
				FB_MC2_Compact_M_nMC_Home_iState:= 030;
			ELSE
				// Error handling
				IF FB_MC2_Compact_M_nMC_Home_fbMC2_Home.Error THEN
					M_nError(nErrorID:= FB_MC2_Compact_M_nMC_Home_fbMC2_Home.ErrorID);
					M_nMC_Home:= FB_MC2_Compact_M_nMC_Home_fbMC2_Home.ErrorID;
					_sMessage:= 'Axis Home Error';
				ELSE
					// Done
					IF FB_MC2_Compact_M_nMC_Home_fbMC2_Home.Done THEN
						FB_MC2_Compact_M_nMC_Home_iState:= 030;
					END_IF
				END_IF
			END_IF
			
	020: // Coupled
			M_nMC_Home:= Tc3_HBI_System.cCOUPLED;
			IF NOT FB_MC2_Compact_M_nMC_Home_bExecute THEN
				FB_MC2_Compact_M_nMC_Home_fbMC2_Halt(Axis:= _stAXIS_REF, Execute:= FALSE); 
				FB_MC2_Compact_M_nMC_Home_fbMC2_Home(Axis:= _stAXIS_REF, Execute:= FALSE);
				FB_MC2_Compact_M_nMC_Home_iState:= 000;
			END_IF

	030:	// Done	
			M_nMC_Home:= Tc3_HBI_System.cCOMPLETE;
			
			IF FB_MC2_Compact_M_nMC_Home_bExecute THEN
				IF FB_MC2_Compact_M_nMC_Home_fbMC2_Halt.CommandAborted OR FB_MC2_Compact_M_nMC_Home_fbMC2_Home.CommandAborted THEN
					M_nMC_Home:= Tc3_HBI_System.cABORTED;
				END_IF
			ELSE
				FB_MC2_Compact_M_nMC_Home_fbMC2_Halt(Axis:= _stAXIS_REF, Execute:= FALSE); 
				FB_MC2_Compact_M_nMC_Home_fbMC2_Home(Axis:= _stAXIS_REF, Execute:= FALSE);
				FB_MC2_Compact_M_nMC_Home_iState:= 000;
			END_IF
		
ELSE
	FB_MC2_Compact_M_nMC_Home_iState:= 000;
END_CASE
END_METHOD

//	The result of the method is an unsigned double integer
//	0 = idle 
//	1 = coupled
//	2 = starting
//	3 = running
//	4 = aborted
// 	5 = no hardware connected
// 	6 = Spare
//	7 = pointer or index error
//	8 = mapping error
//	9 = parameter error
//	10 = complete
//	Any other number = ErrorID
METHOD PUBLIC M_nMC_HomeReset : UDINT
VAR_INPUT
	bExecute: BOOL;
END_VAR
// Local variable
FB_MC2_Compact_M_nMC_HomeReset_bExecute:= bExecute;

//**********************************
// Reset 
//**********************************
IF _bReset THEN
	IF _bError THEN
		FB_MC2_Compact_M_nMC_HomeReset_fbMC2_Home(Axis:= _stAXIS_REF, Execute:= FALSE);
		FB_MC2_Compact_M_nMC_HomeReset_iState:= 000;
		_sMessage:= '';
	END_IF
END_IF

//**********************************
// Wait for execute
//**********************************
IF _stAXIS_REF.NcToPlc.AxisID > 0 THEN
	FB_MC2_Compact_M_nMC_HomeReset_fbExecute_R_TRIG(CLK:= FB_MC2_Compact_M_nMC_HomeReset_bExecute);
	IF FB_MC2_Compact_M_nMC_HomeReset_fbExecute_R_TRIG.Q THEN
		FB_MC2_Compact_M_nMC_HomeReset_fbMC2_Home(Axis:= _stAXIS_REF, Execute:= FALSE, Position:= 0.0, HomingMode:= Tc2_MC2.MC_ResetCalibration, BufferMode:= MC_Aborting, bCalibrationCam:= FALSE);
	
		// Axis not coupled	
		IF NOT _stAXIS_REF.Status.Coupled THEN
			FB_MC2_Compact_M_nMC_HomeReset_iState:= 001;
		ELSE
			FB_MC2_Compact_M_nMC_HomeReset_iState:= 020;
		END_IF
		
	END_IF
ELSE
	FB_MC2_Compact_M_nMC_HomeReset_fbExecute_R_TRIG(CLK:= FALSE);
	FB_MC2_Compact_M_nMC_HomeReset_iState:= 000;
	IF FB_MC2_Compact_M_nMC_HomeReset_bExecute THEN
		M_nMC_HomeReset:= Tc3_HBI_System.cMAPPING_ERROR;
	END_IF
	RETURN;
END_IF


//**********************************
// Main sequence
//**********************************
CASE FB_MC2_Compact_M_nMC_HomeReset_iState OF

	000: 	// Do nothing

	001:	// Home axis
			M_nMC_HomeReset:= Tc3_HBI_System.cRUNNING;
			FB_MC2_Compact_M_nMC_HomeReset_fbMC2_Home(Axis:= _stAXIS_REF, Execute:= TRUE, Position:= 0.0, HomingMode:= Tc2_MC2.MC_ResetCalibration, BufferMode:= MC_Aborting, bCalibrationCam:= FALSE);
		
			// Command aborted
			IF FB_MC2_Compact_M_nMC_HomeReset_fbMC2_Home.CommandAborted THEN
				FB_MC2_Compact_M_nMC_HomeReset_iState:= 030;
			ELSE
				// Error handling
				IF FB_MC2_Compact_M_nMC_HomeReset_fbMC2_Home.Error THEN
					M_nError(nErrorID:= FB_MC2_Compact_M_nMC_HomeReset_fbMC2_Home.ErrorID);
					M_nMC_HomeReset:= FB_MC2_Compact_M_nMC_HomeReset_fbMC2_Home.ErrorID;
					_sMessage:= 'Axis Home Reset Error';
				ELSE
					// Done
					IF FB_MC2_Compact_M_nMC_HomeReset_fbMC2_Home.Done THEN
						FB_MC2_Compact_M_nMC_HomeReset_iState:= 030;
					END_IF
				END_IF
			END_IF
		
	020: // Coupled
			M_nMC_HomeReset:= Tc3_HBI_System.cCOUPLED;
			IF NOT FB_MC2_Compact_M_nMC_HomeReset_bExecute THEN
				FB_MC2_Compact_M_nMC_HomeReset_fbMC2_Home(Axis:= _stAXIS_REF, Execute:= FALSE);
				FB_MC2_Compact_M_nMC_HomeReset_iState:= 000;
			END_IF

	030:	// Done	
			M_nMC_HomeReset:= Tc3_HBI_System.cCOMPLETE;
			
			IF FB_MC2_Compact_M_nMC_HomeReset_bExecute THEN
				IF FB_MC2_Compact_M_nMC_HomeReset_fbMC2_Home.CommandAborted THEN
					M_nMC_HomeReset:= Tc3_HBI_System.cABORTED;
				END_IF
			ELSE
				FB_MC2_Compact_M_nMC_HomeReset_fbMC2_Home(Axis:= _stAXIS_REF, Execute:= FALSE);
				FB_MC2_Compact_M_nMC_HomeReset_iState:= 000;
			END_IF
		
ELSE
	FB_MC2_Compact_M_nMC_HomeReset_iState:= 000;
END_CASE
END_METHOD

//	The result of the method is an unsigned double integer
//	0 = idle 
//	1 = coupled
//	2 = starting
//	3 = running
//	4 = aborted
// 	5 = no hardware connected
// 	6 = Spare
//	7 = pointer or index error
//	8 = mapping error
//	9 = parameter error
//	10 = complete
//	Any other number = ErrorID
METHOD PUBLIC M_nMC_Jog : UDINT
VAR_INPUT
	bForward: BOOL;
	bBackwards: BOOL;
	lrVelocity: LREAL;
END_VAR
// Local variable
FB_MC2_Compact_M_nMC_Jog_bForward:= bForward;
FB_MC2_Compact_M_nMC_Jog_bBackwards:= bBackwards;
FB_MC2_Compact_M_nMC_Jog_lrVelocity:= lrVelocity;

//**********************************
// Reset 
//**********************************
IF _bReset THEN
	IF _bError THEN
		FB_MC2_Compact_M_nMC_Jog_fbMC2_Jog1(Axis:= _stAXIS_REF, JogForward:= FALSE, JogBackwards:= FALSE);
		FB_MC2_Compact_M_nMC_Jog_fbMC2_Jog2(Axis:= _stAXIS_REF, JogForward:= FALSE, JogBackwards:= FALSE);
		FB_MC2_Compact_M_nMC_Jog_iState:= 000;
		_sMessage:= '';
	END_IF	
END_IF

//**********************************
// Parameter check 
//**********************************
IF FB_MC2_Compact_M_nMC_Jog_bForward AND FB_MC2_Compact_M_nMC_Jog_bBackwards THEN
	FB_MC2_Compact_M_nMC_Jog_fbMC2_Jog1(Axis:= _stAXIS_REF, JogForward:= FALSE, JogBackwards:= FALSE);
	FB_MC2_Compact_M_nMC_Jog_fbMC2_Jog2(Axis:= _stAXIS_REF, JogForward:= FALSE, JogBackwards:= FALSE);
	FB_MC2_Compact_M_nMC_Jog_fbExecute_R_TRIG1(CLK:= FALSE);
	FB_MC2_Compact_M_nMC_Jog_fbExecute_R_TRIG2(CLK:= FALSE);
	M_nMC_Jog:= Tc3_HBI_System.cIDLE;
	FB_MC2_Compact_M_nMC_Jog_iState:= 000;
	RETURN;
ELSE
	IF FB_MC2_Compact_M_nMC_Jog_bForward OR FB_MC2_Compact_M_nMC_Jog_bBackwards THEN
		IF _stAXIS_REF.NcToPlc.AxisID = 0 THEN
			FB_MC2_Compact_M_nMC_Jog_fbMC2_Jog1(Axis:= _stAXIS_REF, JogForward:= FALSE, JogBackwards:= FALSE);
			FB_MC2_Compact_M_nMC_Jog_fbMC2_Jog2(Axis:= _stAXIS_REF, JogForward:= FALSE, JogBackwards:= FALSE);
			FB_MC2_Compact_M_nMC_Jog_fbExecute_R_TRIG1(CLK:= FALSE);
			FB_MC2_Compact_M_nMC_Jog_fbExecute_R_TRIG2(CLK:= FALSE);
			M_nMC_Jog:= Tc3_HBI_System.cMAPPING_ERROR;
			FB_MC2_Compact_M_nMC_Jog_iState:= 000;
			RETURN;
		ELSE
			IF FB_MC2_Compact_M_nMC_Jog_lrVelocity <= 0.0 THEN
				FB_MC2_Compact_M_nMC_Jog_fbMC2_Jog1(Axis:= _stAXIS_REF, JogForward:= FALSE, JogBackwards:= FALSE);
				FB_MC2_Compact_M_nMC_Jog_fbMC2_Jog2(Axis:= _stAXIS_REF, JogForward:= FALSE, JogBackwards:= FALSE);
				FB_MC2_Compact_M_nMC_Jog_fbExecute_R_TRIG1(CLK:= FALSE);
				FB_MC2_Compact_M_nMC_Jog_fbExecute_R_TRIG2(CLK:= FALSE);
				M_nMC_Jog:= Tc3_HBI_System.cPARAMETER_ERROR;
				FB_MC2_Compact_M_nMC_Jog_iState:= 000;
				RETURN;
			END_IF
		END_IF
	END_IF
END_IF


//**********************************
// Wait for execute
//**********************************
FB_MC2_Compact_M_nMC_Jog_fbExecute_R_TRIG1(CLK:= FB_MC2_Compact_M_nMC_Jog_bForward);
FB_MC2_Compact_M_nMC_Jog_fbExecute_R_TRIG2(CLK:= FB_MC2_Compact_M_nMC_Jog_bBackwards);
IF FB_MC2_Compact_M_nMC_Jog_fbExecute_R_TRIG1.Q OR FB_MC2_Compact_M_nMC_Jog_fbExecute_R_TRIG2.Q THEN
		FB_MC2_Compact_M_nMC_Jog_fbMC2_Jog1(Axis:= _stAXIS_REF, Mode:= MC_JOGMODE_CONTINOUS, Velocity:= FB_MC2_Compact_M_nMC_Jog_lrVelocity, Acceleration:= _stDynamic.lrAcceleration, Deceleration:= _stDynamic.lrDeceleration, Jerk:= _stDynamic.lrJerk); 
		FB_MC2_Compact_M_nMC_Jog_fbMC2_Jog2(Axis:= _stAXIS_REF, Mode:= MC_JOGMODE_CONTINOUS, Velocity:= FB_MC2_Compact_M_nMC_Jog_lrVelocity, Acceleration:= _stDynamic.lrAcceleration, Deceleration:= _stDynamic.lrDeceleration, Jerk:= _stDynamic.lrJerk); 

		// Axis not coupled	
		IF NOT _stAXIS_REF.Status.Coupled THEN
			IF (FB_MC2_Compact_M_nMC_Jog_fbMC2_Jog1.JogForward OR FB_MC2_Compact_M_nMC_Jog_fbMC2_Jog1.JogBackwards) OR FB_MC2_Compact_M_nMC_Jog_fbMC2_Jog1.Busy THEN
				FB_MC2_Compact_M_nMC_Jog_fbMC2_Jog1(Axis:= _stAXIS_REF, JogForward:= FALSE, JogBackwards:= FALSE);
				FB_MC2_Compact_M_nMC_Jog_fbMC2_Jog2(Axis:= _stAXIS_REF, JogForward:= FALSE, JogBackwards:= FALSE);
				FB_MC2_Compact_M_nMC_Jog_fbMC2_Jog2(Axis:= _stAXIS_REF, JogForward:= FB_MC2_Compact_M_nMC_Jog_bForward, JogBackwards:= FB_MC2_Compact_M_nMC_Jog_bBackwards); 
				FB_MC2_Compact_M_nMC_Jog_iState:= 010;
			ELSE
				FB_MC2_Compact_M_nMC_Jog_fbMC2_Jog1(Axis:= _stAXIS_REF, JogForward:= FALSE, JogBackwards:= FALSE);
				FB_MC2_Compact_M_nMC_Jog_fbMC2_Jog2(Axis:= _stAXIS_REF, JogForward:= FALSE, JogBackwards:= FALSE);
				FB_MC2_Compact_M_nMC_Jog_fbMC2_Jog1(Axis:= _stAXIS_REF, JogForward:= FB_MC2_Compact_M_nMC_Jog_bForward, JogBackwards:= FB_MC2_Compact_M_nMC_Jog_bBackwards);
				FB_MC2_Compact_M_nMC_Jog_iState:= 001;
			END_IF
		ELSE
			FB_MC2_Compact_M_nMC_Jog_fbMC2_Jog1(Axis:= _stAXIS_REF, JogForward:= FALSE, JogBackwards:= FALSE);
			FB_MC2_Compact_M_nMC_Jog_fbMC2_Jog2(Axis:= _stAXIS_REF, JogForward:= FALSE, JogBackwards:= FALSE);
			FB_MC2_Compact_M_nMC_Jog_iState:= 030;
		END_IF
	
END_IF


//**********************************
// Main sequence
//**********************************
CASE FB_MC2_Compact_M_nMC_Jog_iState OF

	000:	// Do nothing

	001:	// Jog1 active
			M_nMC_Jog:= Tc3_HBI_System.cSTARTING;
			FB_MC2_Compact_M_nMC_Jog_fbMC2_Jog1(Axis:= _stAXIS_REF);
			FB_MC2_Compact_M_nMC_Jog_fbMC2_Jog2(Axis:= _stAXIS_REF);
			
			// Command aborted
			IF FB_MC2_Compact_M_nMC_Jog_fbMC2_Jog1.CommandAborted THEN
				FB_MC2_Compact_M_nMC_Jog_fbMC2_Jog2.JogForward:= FALSE; 
				FB_MC2_Compact_M_nMC_Jog_fbMC2_Jog2.JogBackwards:= FALSE; 
				FB_MC2_Compact_M_nMC_Jog_iState:= 040;
			ELSE
				// Error handling
				IF FB_MC2_Compact_M_nMC_Jog_fbMC2_Jog1.Error THEN
					M_nError(nErrorID:= FB_MC2_Compact_M_nMC_Jog_fbMC2_Jog1.ErrorID);
					M_nMC_Jog:= FB_MC2_Compact_M_nMC_Jog_fbMC2_Jog1.ErrorID;
					_sMessage:= 'Axis Jog Error';
				ELSE
					// Active
					IF FB_MC2_Compact_M_nMC_Jog_fbMC2_Jog1.Active THEN
						FB_MC2_Compact_M_nMC_Jog_iState:= 002;
					ELSE
						// Done
						IF NOT FB_MC2_Compact_M_nMC_Jog_bForward AND NOT FB_MC2_Compact_M_nMC_Jog_bBackwards THEN
							FB_MC2_Compact_M_nMC_Jog_iState:= 040;
						END_IF
					END_IF	
				END_IF
			END_IF
		
	002:	// Jog1 done
			FB_MC2_Compact_M_nMC_Jog_fbMC2_Jog1(Axis:= _stAXIS_REF); 
			FB_MC2_Compact_M_nMC_Jog_fbMC2_Jog2(Axis:= _stAXIS_REF); 
			
			// Command aborted
			IF FB_MC2_Compact_M_nMC_Jog_fbMC2_Jog1.CommandAborted THEN
				FB_MC2_Compact_M_nMC_Jog_fbMC2_Jog2.JogForward:= FALSE; 
				FB_MC2_Compact_M_nMC_Jog_fbMC2_Jog2.JogBackwards:= FALSE; 
				FB_MC2_Compact_M_nMC_Jog_iState:= 040;
			ELSE
				// Error handling
				IF FB_MC2_Compact_M_nMC_Jog_fbMC2_Jog1.Error THEN
					M_nError(nErrorID:= FB_MC2_Compact_M_nMC_Jog_fbMC2_Jog1.ErrorID);
					M_nMC_Jog:= FB_MC2_Compact_M_nMC_Jog_fbMC2_Jog1.ErrorID;
					_sMessage:= 'Axis Jog Error';
				ELSE
					// Done
					IF NOT FB_MC2_Compact_M_nMC_Jog_bForward AND NOT FB_MC2_Compact_M_nMC_Jog_bBackwards THEN
						FB_MC2_Compact_M_nMC_Jog_iState:= 040;
					END_IF	
				END_IF
			END_IF

			// Done
			IF _stAXIS_REF.Status.ConstantVelocity THEN
				M_nMC_Jog:= Tc3_HBI_System.cCOMPLETE;
			ELSE
				M_nMC_Jog:= Tc3_HBI_System.cRUNNING;
			END_IF
	
	010:	// Jog2 active 
			M_nMC_Jog:= Tc3_HBI_System.cSTARTING;
			FB_MC2_Compact_M_nMC_Jog_fbMC2_Jog1(Axis:= _stAXIS_REF); 
			FB_MC2_Compact_M_nMC_Jog_fbMC2_Jog2(Axis:= _stAXIS_REF); 

			// Command aborted
			IF FB_MC2_Compact_M_nMC_Jog_fbMC2_Jog2.CommandAborted THEN
				FB_MC2_Compact_M_nMC_Jog_fbMC2_Jog1.JogForward:= FALSE; 
				FB_MC2_Compact_M_nMC_Jog_fbMC2_Jog1.JogBackwards:= FALSE; 
				FB_MC2_Compact_M_nMC_Jog_iState:= 040;
			ELSE
				// Error handling
				IF FB_MC2_Compact_M_nMC_Jog_fbMC2_Jog2.Error THEN
					M_nError(nErrorID:= FB_MC2_Compact_M_nMC_Jog_fbMC2_Jog2.ErrorID);
					M_nMC_Jog:= FB_MC2_Compact_M_nMC_Jog_fbMC2_Jog2.ErrorID;
					_sMessage:= 'Axis Jog Error';
				ELSE
					// Active
					IF FB_MC2_Compact_M_nMC_Jog_fbMC2_Jog2.Active THEN
						FB_MC2_Compact_M_nMC_Jog_iState:= 011;
					ELSE
						// Done
						IF NOT FB_MC2_Compact_M_nMC_Jog_bForward AND NOT FB_MC2_Compact_M_nMC_Jog_bBackwards THEN
							FB_MC2_Compact_M_nMC_Jog_iState:= 040;
						END_IF
					END_IF	
				END_IF
			END_IF

	011:	// Jog2 done
			M_nMC_Jog:= Tc3_HBI_System.cRUNNING;
			FB_MC2_Compact_M_nMC_Jog_fbMC2_Jog1(Axis:= _stAXIS_REF); 
			FB_MC2_Compact_M_nMC_Jog_fbMC2_Jog2(Axis:= _stAXIS_REF); 
			
			// Command aborted
			IF FB_MC2_Compact_M_nMC_Jog_fbMC2_Jog2.CommandAborted THEN
				FB_MC2_Compact_M_nMC_Jog_fbMC2_Jog1.JogForward:= FALSE; 
				FB_MC2_Compact_M_nMC_Jog_fbMC2_Jog1.JogBackwards:= FALSE; 
				FB_MC2_Compact_M_nMC_Jog_iState:= 040;
			ELSE
				// Error handling
				IF FB_MC2_Compact_M_nMC_Jog_fbMC2_Jog2.Error THEN
					M_nError(nErrorID:= FB_MC2_Compact_M_nMC_Jog_fbMC2_Jog2.ErrorID);
					M_nMC_Jog:= FB_MC2_Compact_M_nMC_Jog_fbMC2_Jog2.ErrorID;
					_sMessage:= 'Axis Jog Error';
				ELSE
					// Done
					IF NOT FB_MC2_Compact_M_nMC_Jog_bForward AND NOT FB_MC2_Compact_M_nMC_Jog_bBackwards THEN
						FB_MC2_Compact_M_nMC_Jog_iState:= 040;
					END_IF	
				END_IF	
			END_IF
	
			// Done
			IF _stAXIS_REF.Status.ConstantVelocity THEN
				M_nMC_Jog:= Tc3_HBI_System.cCOMPLETE;
			ELSE
				M_nMC_Jog:= Tc3_HBI_System.cRUNNING;
			END_IF
			
	030: // Coupled
			M_nMC_Jog:= Tc3_HBI_System.cCOUPLED;
			FB_MC2_Compact_M_nMC_Jog_fbMC2_Jog1(Axis:= _stAXIS_REF); 
			FB_MC2_Compact_M_nMC_Jog_fbMC2_Jog2(Axis:= _stAXIS_REF); 

			IF NOT FB_MC2_Compact_M_nMC_Jog_bForward AND NOT FB_MC2_Compact_M_nMC_Jog_bBackwards THEN
				FB_MC2_Compact_M_nMC_Jog_fbMC2_Jog1(Axis:= _stAXIS_REF, JogForward:= FALSE, JogBackwards:= FALSE);
				FB_MC2_Compact_M_nMC_Jog_fbMC2_Jog2(Axis:= _stAXIS_REF, JogForward:= FALSE, JogBackwards:= FALSE);
				FB_MC2_Compact_M_nMC_Jog_iState:= 000;
			END_IF

	040:	// Done
			FB_MC2_Compact_M_nMC_Jog_fbMC2_Jog1(Axis:= _stAXIS_REF, JogForward:= FB_MC2_Compact_M_nMC_Jog_bForward, JogBackwards:= bBackwards);
			FB_MC2_Compact_M_nMC_Jog_fbMC2_Jog2(Axis:= _stAXIS_REF, JogForward:= FB_MC2_Compact_M_nMC_Jog_bForward, JogBackwards:= bBackwards);

			// Status
			IF _stAXIS_REF.Status.HasJob AND _stAXIS_REF.Status.Moving THEN
				M_nMC_Jog:= Tc3_HBI_System.cRUNNING;
			ELSE
				M_nMC_Jog:= Tc3_HBI_System.cCOMPLETE;
				FB_MC2_Compact_M_nMC_Jog_fbMC2_Jog1(Axis:= _stAXIS_REF, JogForward:= FALSE, JogBackwards:= FALSE);
				FB_MC2_Compact_M_nMC_Jog_fbMC2_Jog2(Axis:= _stAXIS_REF, JogForward:= FALSE, JogBackwards:= FALSE);
				FB_MC2_Compact_M_nMC_Jog_iState:= 000;
			END_IF
			
			IF FB_MC2_Compact_M_nMC_Jog_bForward OR FB_MC2_Compact_M_nMC_Jog_bBackwards THEN
				IF (FB_MC2_Compact_M_nMC_Jog_fbMC2_Jog1.JogForward OR FB_MC2_Compact_M_nMC_Jog_fbMC2_Jog1.JogBackwards) AND FB_MC2_Compact_M_nMC_Jog_fbMC2_Jog1.CommandAborted THEN
					M_nMC_Jog:= Tc3_HBI_System.cABORTED;
				END_IF
				IF (FB_MC2_Compact_M_nMC_Jog_fbMC2_Jog2.JogForward OR FB_MC2_Compact_M_nMC_Jog_fbMC2_Jog2.JogBackwards) AND FB_MC2_Compact_M_nMC_Jog_fbMC2_Jog2.CommandAborted THEN
					M_nMC_Jog:= Tc3_HBI_System.cABORTED;
				END_IF
			END_IF

ELSE
	FB_MC2_Compact_M_nMC_Jog_iState:= 000;
END_CASE
END_METHOD

//	The result of the method is an unsigned double integer
//	0 = idle 
//	1 = coupled
//	2 = starting
//	3 = running
//	4 = aborted
// 	5 = no hardware connected
// 	6 = Spare
//	7 = pointer or index error
//	8 = mapping error
//	9 = parameter error
//	10 = complete
//	Any other number = ErrorID
METHOD PRIVATE M_nMC_Local_Halt : UDINT
VAR_INPUT
	bExecute: BOOL;
END_VAR
// Local variable
FB_MC2_Compact_M_nMC_Local_Halt_bExecute:= bExecute;

//**********************************
// Reset 
//**********************************
IF _bReset THEN
	IF _bError THEN
		FB_MC2_Compact_M_nMC_Local_Halt_fbMC2_Halt1(Axis:= _stAXIS_REF, Execute:= FALSE);
		FB_MC2_Compact_M_nMC_Local_Halt_fbMC2_Halt2(Axis:= _stAXIS_REF, Execute:= FALSE);
		FB_MC2_Compact_M_nMC_Local_Halt_iState:= 000;
		_sMessage:= '';
	END_IF
END_IF

//**********************************
// Wait for execute
//**********************************
IF _stAXIS_REF.NcToPlc.AxisID > 0 THEN
	FB_MC2_Compact_M_nMC_Local_Halt_fbExecute_R_TRIG(CLK:= FB_MC2_Compact_M_nMC_Local_Halt_bExecute);
	IF FB_MC2_Compact_M_nMC_Local_Halt_fbExecute_R_TRIG.Q THEN
			FB_MC2_Compact_M_nMC_Local_Halt_fbMC2_Halt1(Axis:= _stAXIS_REF, Deceleration:= _stDynamic.lrDeceleration, Jerk:= _stDynamic.lrJerk, BufferMode:= _eBufferMode);
			FB_MC2_Compact_M_nMC_Local_Halt_fbMC2_Halt2(Axis:= _stAXIS_REF, Deceleration:= _stDynamic.lrDeceleration, Jerk:= _stDynamic.lrJerk, BufferMode:= _eBufferMode);
	
			// Axis not coupled	
			IF NOT _stAXIS_REF.Status.Coupled THEN
				IF _stAXIS_REF.Status.ControlLoopClosed THEN
					IF _stAXIS_REF.Status.HasJob THEN
						IF FB_MC2_Compact_M_nMC_Local_Halt_fbMC2_Halt1.Execute OR FB_MC2_Compact_M_nMC_Local_Halt_fbMC2_Halt1.Busy THEN
							FB_MC2_Compact_M_nMC_Local_Halt_fbMC2_Halt1(Axis:= _stAXIS_REF, Execute:= FALSE);
							FB_MC2_Compact_M_nMC_Local_Halt_fbMC2_Halt2(Axis:= _stAXIS_REF, Execute:= FALSE);
							FB_MC2_Compact_M_nMC_Local_Halt_fbMC2_Halt2.Execute:= TRUE;
							FB_MC2_Compact_M_nMC_Local_Halt_iState:= 010;
						ELSE
							FB_MC2_Compact_M_nMC_Local_Halt_fbMC2_Halt1(Axis:= _stAXIS_REF, Execute:= FALSE);
							FB_MC2_Compact_M_nMC_Local_Halt_fbMC2_Halt2(Axis:= _stAXIS_REF, Execute:= FALSE);
							FB_MC2_Compact_M_nMC_Local_Halt_fbMC2_Halt1.Execute:= TRUE;
							FB_MC2_Compact_M_nMC_Local_Halt_iState:= 001;
						END_IF
					ELSE
						FB_MC2_Compact_M_nMC_Local_Halt_iState:= 040;
					END_IF	
				ELSE
					FB_MC2_Compact_M_nMC_Local_Halt_iState:= 040;
				END_IF	
			ELSE
				FB_MC2_Compact_M_nMC_Local_Halt_fbMC2_Halt1(Axis:= _stAXIS_REF, Execute:= FALSE);
				FB_MC2_Compact_M_nMC_Local_Halt_fbMC2_Halt2(Axis:= _stAXIS_REF, Execute:= FALSE);
				FB_MC2_Compact_M_nMC_Local_Halt_iState:= 030;
			END_IF
		
	END_IF
ELSE
	FB_MC2_Compact_M_nMC_Local_Halt_fbExecute_R_TRIG(CLK:= FALSE);
	FB_MC2_Compact_M_nMC_Local_Halt_iState:= 000;
	IF FB_MC2_Compact_M_nMC_Local_Halt_bExecute THEN
		M_nMC_Local_Halt:= Tc3_HBI_System.cMAPPING_ERROR;
	END_IF
	RETURN;
END_IF


//**********************************
// Main sequence
//**********************************
CASE FB_MC2_Compact_M_nMC_Local_Halt_iState OF

	000: 	// Do nothing
	
	001:	// Stop Axis1
			M_nMC_Local_Halt:= Tc3_HBI_System.cSTARTING;
			FB_MC2_Compact_M_nMC_Local_Halt_fbMC2_Halt1(Axis:= _stAXIS_REF);
			FB_MC2_Compact_M_nMC_Local_Halt_fbMC2_Halt2(Axis:= _stAXIS_REF);
	
			// Command aborted
			IF FB_MC2_Compact_M_nMC_Local_Halt_fbMC2_Halt1.CommandAborted THEN
				FB_MC2_Compact_M_nMC_Local_Halt_fbMC2_Halt2.Execute:= FALSE;
				FB_MC2_Compact_M_nMC_Local_Halt_iState:= 040;
			ELSE
				// Error handling
				IF FB_MC2_Compact_M_nMC_Local_Halt_fbMC2_Halt1.Error THEN
					M_nError(FB_MC2_Compact_M_nMC_Local_Halt_fbMC2_Halt1.ErrorID);
					M_nMC_Local_Halt:= FB_MC2_Compact_M_nMC_Local_Halt_fbMC2_Halt1.ErrorID;
					_sMessage:= 'Axis Local Halt Error';
				ELSE
					// Active
					IF FB_MC2_Compact_M_nMC_Local_Halt_fbMC2_Halt1.Active THEN
						FB_MC2_Compact_M_nMC_Local_Halt_iState:= 002;
					ELSE
						// Done
						IF FB_MC2_Compact_M_nMC_Local_Halt_fbMC2_Halt1.Done THEN
							FB_MC2_Compact_M_nMC_Local_Halt_iState:= 040;
						END_IF
					END_IF	
				END_IF
			END_IF

	002:	// Stop Axis
			M_nMC_Local_Halt:= Tc3_HBI_System.cRUNNING;
			FB_MC2_Compact_M_nMC_Local_Halt_fbMC2_Halt1(Axis:= _stAXIS_REF);
			FB_MC2_Compact_M_nMC_Local_Halt_fbMC2_Halt2(Axis:= _stAXIS_REF);
	
			// Command aborted
			IF FB_MC2_Compact_M_nMC_Local_Halt_fbMC2_Halt1.CommandAborted THEN
				FB_MC2_Compact_M_nMC_Local_Halt_fbMC2_Halt2.Execute:= FALSE;
				FB_MC2_Compact_M_nMC_Local_Halt_iState:= 040;
			ELSE
				// Error handling
				IF FB_MC2_Compact_M_nMC_Local_Halt_fbMC2_Halt1.Error THEN
					M_nError(FB_MC2_Compact_M_nMC_Local_Halt_fbMC2_Halt1.ErrorID);
					M_nMC_Local_Halt:= FB_MC2_Compact_M_nMC_Local_Halt_fbMC2_Halt1.ErrorID;
					_sMessage:= 'Axis Local Halt Error';
				ELSE
					// Done
					IF FB_MC2_Compact_M_nMC_Local_Halt_fbMC2_Halt1.Done THEN
						FB_MC2_Compact_M_nMC_Local_Halt_iState:= 040;
					END_IF
				END_IF
			END_IF 
	
	010:	// Stop Axis1
			M_nMC_Local_Halt:= Tc3_HBI_System.cSTARTING;
			FB_MC2_Compact_M_nMC_Local_Halt_fbMC2_Halt1(Axis:= _stAXIS_REF);
			FB_MC2_Compact_M_nMC_Local_Halt_fbMC2_Halt2(Axis:= _stAXIS_REF);
			
			// Command aborted
			IF FB_MC2_Compact_M_nMC_Local_Halt_fbMC2_Halt2.CommandAborted THEN
				FB_MC2_Compact_M_nMC_Local_Halt_fbMC2_Halt1.Execute:= FALSE;
				FB_MC2_Compact_M_nMC_Local_Halt_iState:= 040;
			ELSE
				// Error handling
				IF FB_MC2_Compact_M_nMC_Local_Halt_fbMC2_Halt2.Error THEN
					M_nError(FB_MC2_Compact_M_nMC_Local_Halt_fbMC2_Halt2.ErrorID);
					M_nMC_Local_Halt:= FB_MC2_Compact_M_nMC_Local_Halt_fbMC2_Halt2.ErrorID;
					_sMessage:= 'Axis Local Halt Error';
				ELSE
					// Active
					IF FB_MC2_Compact_M_nMC_Local_Halt_fbMC2_Halt2.Active THEN
						FB_MC2_Compact_M_nMC_Local_Halt_iState:= 011;
					ELSE
						// Done
						IF FB_MC2_Compact_M_nMC_Local_Halt_fbMC2_Halt2.Done THEN
							FB_MC2_Compact_M_nMC_Local_Halt_iState:= 040;
						END_IF
					END_IF	
				END_IF
			END_IF 
		
	011:	// Stop Axis2
			M_nMC_Local_Halt:= Tc3_HBI_System.cRUNNING;
			FB_MC2_Compact_M_nMC_Local_Halt_fbMC2_Halt1(Axis:= _stAXIS_REF);
			FB_MC2_Compact_M_nMC_Local_Halt_fbMC2_Halt2(Axis:= _stAXIS_REF);
			
			// Command aborted
			IF FB_MC2_Compact_M_nMC_Local_Halt_fbMC2_Halt2.CommandAborted THEN
				FB_MC2_Compact_M_nMC_Local_Halt_fbMC2_Halt1.Execute:= FALSE;
				FB_MC2_Compact_M_nMC_Local_Halt_iState:= 040;
			ELSE
				// Error handling
				IF FB_MC2_Compact_M_nMC_Local_Halt_fbMC2_Halt2.Error THEN
					M_nError(FB_MC2_Compact_M_nMC_Local_Halt_fbMC2_Halt2.ErrorID);
					M_nMC_Local_Halt:= FB_MC2_Compact_M_nMC_Local_Halt_fbMC2_Halt2.ErrorID;
					_sMessage:= 'Axis Local Halt Error';
				ELSE
					// Done
					IF FB_MC2_Compact_M_nMC_Local_Halt_fbMC2_Halt2.Done THEN
						FB_MC2_Compact_M_nMC_Local_Halt_iState:= 040;
					END_IF
				END_IF
			END_IF
	
	030:	// Coupled
			M_nMC_Local_Halt:= Tc3_HBI_System.cCOUPLED;
			FB_MC2_Compact_M_nMC_Local_Halt_fbMC2_Halt1(Axis:= _stAXIS_REF);
			FB_MC2_Compact_M_nMC_Local_Halt_fbMC2_Halt2(Axis:= _stAXIS_REF);

			IF NOT FB_MC2_Compact_M_nMC_Local_Halt_bExecute THEN
				FB_MC2_Compact_M_nMC_Local_Halt_fbMC2_Halt1(Axis:= _stAXIS_REF, Execute:= FALSE);
				FB_MC2_Compact_M_nMC_Local_Halt_fbMC2_Halt2(Axis:= _stAXIS_REF, Execute:= FALSE);
				FB_MC2_Compact_M_nMC_Local_Halt_iState:= 000;
			END_IF	
	
	040:	// Done
			M_nMC_Local_Halt:= Tc3_HBI_System.cCOMPLETE;
			FB_MC2_Compact_M_nMC_Local_Halt_fbMC2_Halt1(Axis:= _stAXIS_REF);
			FB_MC2_Compact_M_nMC_Local_Halt_fbMC2_Halt2(Axis:= _stAXIS_REF);
			
			IF FB_MC2_Compact_M_nMC_Local_Halt_bExecute THEN
				IF FB_MC2_Compact_M_nMC_Local_Halt_fbMC2_Halt1.Execute AND FB_MC2_Compact_M_nMC_Local_Halt_fbMC2_Halt1.CommandAborted THEN
					M_nMC_Local_Halt:= Tc3_HBI_System.cABORTED;
				END_IF
				IF FB_MC2_Compact_M_nMC_Local_Halt_fbMC2_Halt2.Execute AND FB_MC2_Compact_M_nMC_Local_Halt_fbMC2_Halt2.CommandAborted THEN
					M_nMC_Local_Halt:= Tc3_HBI_System.cABORTED;
				END_IF
			ELSE
				FB_MC2_Compact_M_nMC_Local_Halt_fbMC2_Halt1(Axis:= _stAXIS_REF, Execute:= FALSE);
				FB_MC2_Compact_M_nMC_Local_Halt_fbMC2_Halt2(Axis:= _stAXIS_REF, Execute:= FALSE);
				FB_MC2_Compact_M_nMC_Local_Halt_iState:= 000;
			END_IF	
		
ELSE
	FB_MC2_Compact_M_nMC_Local_Halt_iState:= 000;
END_CASE
END_METHOD

//	The result of the method is an unsigned double integer
//	0 = idle 
//	1 = coupled
//	2 = starting
//	3 = running
//	4 = aborted
// 	5 = no hardware connected
// 	6 = Spare
//	7 = pointer or index error
//	8 = mapping error
//	9 = parameter error
//	10 = complete
//	Any other number = ErrorID
METHOD PUBLIC M_nMC_MoveAbsolute : UDINT
VAR_INPUT
	bExecute: BOOL;
	lrPosition: LREAL;
	lrVelocity: LREAL;
END_VAR
// Local variable
FB_MC2_Compact_M_nMC_MoveAbsolute_bExecute:= bExecute;
FB_MC2_Compact_M_nMC_MoveAbsolute_lrPosition:= lrPosition;
FB_MC2_Compact_M_nMC_MoveAbsolute_lrVelocity:= lrVelocity;

//**********************************
// Reset 
//**********************************
IF _bReset THEN
	IF _bError THEN
		FB_MC2_Compact_M_nMC_MoveAbsolute_fbMC2_MoveAbsolute1(Axis:= _stAXIS_REF, Execute:= FALSE);
		FB_MC2_Compact_M_nMC_MoveAbsolute_fbMC2_MoveAbsolute2(Axis:= _stAXIS_REF, Execute:= FALSE);
		FB_MC2_Compact_M_nMC_MoveAbsolute_iState:= 000;
		_sMessage:= '';
	END_IF		
END_IF

//**********************************
// Wait for execute
//**********************************
IF _stAXIS_REF.NcToPlc.AxisID > 0 THEN
	FB_MC2_Compact_M_nMC_MoveAbsolute_fbExecute_R_TRIG(CLK:= FB_MC2_Compact_M_nMC_MoveAbsolute_bExecute);
	IF FB_MC2_Compact_M_nMC_MoveAbsolute_fbExecute_R_TRIG.Q THEN
		FB_MC2_Compact_M_nMC_MoveAbsolute_fbMC2_MoveAbsolute1(Axis:= _stAXIS_REF, Position:= FB_MC2_Compact_M_nMC_MoveAbsolute_lrPosition, Velocity:= FB_MC2_Compact_M_nMC_MoveAbsolute_lrVelocity, Acceleration:= _stDynamic.lrAcceleration, Deceleration:= _stDynamic.lrDeceleration, Jerk:= _stDynamic.lrJerk, BufferMode:= _eBufferMode); 
		FB_MC2_Compact_M_nMC_MoveAbsolute_fbMC2_MoveAbsolute2(Axis:= _stAXIS_REF, Position:= FB_MC2_Compact_M_nMC_MoveAbsolute_lrPosition, Velocity:= FB_MC2_Compact_M_nMC_MoveAbsolute_lrVelocity, Acceleration:= _stDynamic.lrAcceleration, Deceleration:= _stDynamic.lrDeceleration, Jerk:= _stDynamic.lrJerk, BufferMode:= _eBufferMode); 
		
		// Axis not coupled	
		IF NOT _stAXIS_REF.Status.Coupled THEN
			IF FB_MC2_Compact_M_nMC_MoveAbsolute_fbMC2_MoveAbsolute1.Execute OR FB_MC2_Compact_M_nMC_MoveAbsolute_fbMC2_MoveAbsolute1.Busy THEN
				FB_MC2_Compact_M_nMC_MoveAbsolute_fbMC2_MoveAbsolute1(Axis:= _stAXIS_REF, Execute:= FALSE);
				FB_MC2_Compact_M_nMC_MoveAbsolute_fbMC2_MoveAbsolute2(Axis:= _stAXIS_REF, Execute:= FALSE);
				FB_MC2_Compact_M_nMC_MoveAbsolute_fbMC2_MoveAbsolute2.Execute:= TRUE;
				FB_MC2_Compact_M_nMC_MoveAbsolute_iState:= 010;
			ELSE	
				FB_MC2_Compact_M_nMC_MoveAbsolute_fbMC2_MoveAbsolute1(Axis:= _stAXIS_REF, Execute:= FALSE);
				FB_MC2_Compact_M_nMC_MoveAbsolute_fbMC2_MoveAbsolute2(Axis:= _stAXIS_REF, Execute:= FALSE);
				FB_MC2_Compact_M_nMC_MoveAbsolute_fbMC2_MoveAbsolute1.Execute:= TRUE;
				FB_MC2_Compact_M_nMC_MoveAbsolute_iState:= 001;
			END_IF	
		ELSE
			FB_MC2_Compact_M_nMC_MoveAbsolute_fbMC2_MoveAbsolute1(Axis:= _stAXIS_REF, Execute:= FALSE);
			FB_MC2_Compact_M_nMC_MoveAbsolute_fbMC2_MoveAbsolute2(Axis:= _stAXIS_REF, Execute:= FALSE);
			FB_MC2_Compact_M_nMC_MoveAbsolute_iState:= 030;
		END_IF
	
	END_IF
ELSE
	FB_MC2_Compact_M_nMC_MoveAbsolute_fbExecute_R_TRIG(CLK:= FALSE);
	FB_MC2_Compact_M_nMC_MoveAbsolute_iState:= 000;
	IF FB_MC2_Compact_M_nMC_MoveAbsolute_bExecute THEN
		M_nMC_MoveAbsolute:= Tc3_HBI_System.cMAPPING_ERROR;
	END_IF
	RETURN;
END_IF


//**********************************
// Main sequence
//**********************************
CASE FB_MC2_Compact_M_nMC_MoveAbsolute_iState OF

	000:	// Do nothing

	001:	// MoveAbsolute1 active
			M_nMC_MoveAbsolute:= Tc3_HBI_System.cSTARTING;
			FB_MC2_Compact_M_nMC_MoveAbsolute_fbMC2_MoveAbsolute1(Axis:= _stAXIS_REF); 
			FB_MC2_Compact_M_nMC_MoveAbsolute_fbMC2_MoveAbsolute2(Axis:= _stAXIS_REF); 
	
			// Command aborted
			IF FB_MC2_Compact_M_nMC_MoveAbsolute_fbMC2_MoveAbsolute1.CommandAborted THEN
				FB_MC2_Compact_M_nMC_MoveAbsolute_fbMC2_MoveAbsolute2.Execute:= FALSE; 
				FB_MC2_Compact_M_nMC_MoveAbsolute_iState:= 040;
			ELSE
				// Error handling
				IF FB_MC2_Compact_M_nMC_MoveAbsolute_fbMC2_MoveAbsolute1.Error THEN
					M_nError(nErrorID:= FB_MC2_Compact_M_nMC_MoveAbsolute_fbMC2_MoveAbsolute1.ErrorID);
					M_nMC_MoveAbsolute:= FB_MC2_Compact_M_nMC_MoveAbsolute_fbMC2_MoveAbsolute1.ErrorID;
					_sMessage:= 'Axis Move Absolute Error';
				ELSE
					// Active
					IF FB_MC2_Compact_M_nMC_MoveAbsolute_fbMC2_MoveAbsolute1.Active THEN
						FB_MC2_Compact_M_nMC_MoveAbsolute_iState:= 002;
					ELSE
						// Done
						IF FB_MC2_Compact_M_nMC_MoveAbsolute_fbMC2_MoveAbsolute1.Done THEN
							FB_MC2_Compact_M_nMC_MoveAbsolute_iState:= 040;
						END_IF
					END_IF	
				END_IF
			END_IF
		
	002:	// MoveAbsolute1 done
			M_nMC_MoveAbsolute:= Tc3_HBI_System.cRUNNING;
			FB_MC2_Compact_M_nMC_MoveAbsolute_fbMC2_MoveAbsolute1(Axis:= _stAXIS_REF); 
			FB_MC2_Compact_M_nMC_MoveAbsolute_fbMC2_MoveAbsolute2(Axis:= _stAXIS_REF); 
	
			// Command aborted
			IF FB_MC2_Compact_M_nMC_MoveAbsolute_fbMC2_MoveAbsolute1.CommandAborted THEN
				FB_MC2_Compact_M_nMC_MoveAbsolute_fbMC2_MoveAbsolute2.Execute:= FALSE; 			
				FB_MC2_Compact_M_nMC_MoveAbsolute_iState:= 040;
			ELSE
				// Error handling
				IF FB_MC2_Compact_M_nMC_MoveAbsolute_fbMC2_MoveAbsolute1.Error THEN
					M_nError(nErrorID:= FB_MC2_Compact_M_nMC_MoveAbsolute_fbMC2_MoveAbsolute1.ErrorID);
					M_nMC_MoveAbsolute:= FB_MC2_Compact_M_nMC_MoveAbsolute_fbMC2_MoveAbsolute1.ErrorID;
					_sMessage:= 'Axis Move Absolute Error';
				ELSE
					// Done
					IF FB_MC2_Compact_M_nMC_MoveAbsolute_fbMC2_MoveAbsolute1.Done THEN
						FB_MC2_Compact_M_nMC_MoveAbsolute_iState:= 040;
					END_IF	
				END_IF
			END_IF
	
	010:	// Call MoveAbsolute2 active 
			M_nMC_MoveAbsolute:= Tc3_HBI_System.cSTARTING;
			FB_MC2_Compact_M_nMC_MoveAbsolute_fbMC2_MoveAbsolute1(Axis:= _stAXIS_REF); 
			FB_MC2_Compact_M_nMC_MoveAbsolute_fbMC2_MoveAbsolute2(Axis:= _stAXIS_REF); 
		
			// Command aborted
			IF FB_MC2_Compact_M_nMC_MoveAbsolute_fbMC2_MoveAbsolute2.CommandAborted THEN
				FB_MC2_Compact_M_nMC_MoveAbsolute_fbMC2_MoveAbsolute1.Execute:= FALSE; 
				FB_MC2_Compact_M_nMC_MoveAbsolute_iState:= 040;
			ELSE
				// Error handling
				IF FB_MC2_Compact_M_nMC_MoveAbsolute_fbMC2_MoveAbsolute2.Error THEN
					M_nError(nErrorID:= FB_MC2_Compact_M_nMC_MoveAbsolute_fbMC2_MoveAbsolute2.ErrorID);
					M_nMC_MoveAbsolute:= FB_MC2_Compact_M_nMC_MoveAbsolute_fbMC2_MoveAbsolute2.ErrorID;
					_sMessage:= 'Axis Move Absolute Error';
				ELSE
					// Active
					IF FB_MC2_Compact_M_nMC_MoveAbsolute_fbMC2_MoveAbsolute2.Active THEN
						FB_MC2_Compact_M_nMC_MoveAbsolute_iState:= 011;
					ELSE
						// Done
						IF FB_MC2_Compact_M_nMC_MoveAbsolute_fbMC2_MoveAbsolute2.Done THEN
							FB_MC2_Compact_M_nMC_MoveAbsolute_iState:= 040;
						END_IF
					END_IF	
				END_IF
			END_IF

	011:	// MoveAbsolute2 done
			M_nMC_MoveAbsolute:= Tc3_HBI_System.cRUNNING;
			FB_MC2_Compact_M_nMC_MoveAbsolute_fbMC2_MoveAbsolute1(Axis:= _stAXIS_REF); 
			FB_MC2_Compact_M_nMC_MoveAbsolute_fbMC2_MoveAbsolute2(Axis:= _stAXIS_REF); 
			
			// Command aborted
			IF FB_MC2_Compact_M_nMC_MoveAbsolute_fbMC2_MoveAbsolute2.CommandAborted THEN
				FB_MC2_Compact_M_nMC_MoveAbsolute_fbMC2_MoveAbsolute1.Execute:= FALSE; 
				FB_MC2_Compact_M_nMC_MoveAbsolute_iState:= 040;
			ELSE
				// Error handling
				IF FB_MC2_Compact_M_nMC_MoveAbsolute_fbMC2_MoveAbsolute2.Error THEN
					M_nError(nErrorID:= FB_MC2_Compact_M_nMC_MoveAbsolute_fbMC2_MoveAbsolute2.ErrorID);
					M_nMC_MoveAbsolute:= FB_MC2_Compact_M_nMC_MoveAbsolute_fbMC2_MoveAbsolute2.ErrorID;
					_sMessage:= 'Axis Move Absolute Error';
				ELSE
					// Done
					IF FB_MC2_Compact_M_nMC_MoveAbsolute_fbMC2_MoveAbsolute2.Done THEN
						FB_MC2_Compact_M_nMC_MoveAbsolute_iState:= 040;
					END_IF	
				END_IF	
			END_IF
	
	030: // Coupled
			M_nMC_MoveAbsolute:= Tc3_HBI_System.cCOUPLED;
			FB_MC2_Compact_M_nMC_MoveAbsolute_fbMC2_MoveAbsolute1(Axis:= _stAXIS_REF); 
			FB_MC2_Compact_M_nMC_MoveAbsolute_fbMC2_MoveAbsolute2(Axis:= _stAXIS_REF); 

			IF NOT FB_MC2_Compact_M_nMC_MoveAbsolute_bExecute THEN
				FB_MC2_Compact_M_nMC_MoveAbsolute_fbMC2_MoveAbsolute1(Axis:= _stAXIS_REF, Execute:= FALSE);
				FB_MC2_Compact_M_nMC_MoveAbsolute_fbMC2_MoveAbsolute2(Axis:= _stAXIS_REF, Execute:= FALSE);
				FB_MC2_Compact_M_nMC_MoveAbsolute_iState:= 000;
			END_IF

	040:	// Done
			M_nMC_MoveAbsolute:= Tc3_HBI_System.cCOMPLETE;
			FB_MC2_Compact_M_nMC_MoveAbsolute_fbMC2_MoveAbsolute1(Axis:= _stAXIS_REF); 
			FB_MC2_Compact_M_nMC_MoveAbsolute_fbMC2_MoveAbsolute2(Axis:= _stAXIS_REF); 

			IF FB_MC2_Compact_M_nMC_MoveAbsolute_bExecute THEN
				IF FB_MC2_Compact_M_nMC_MoveAbsolute_fbMC2_MoveAbsolute1.Execute AND FB_MC2_Compact_M_nMC_MoveAbsolute_fbMC2_MoveAbsolute1.CommandAborted THEN
					M_nMC_MoveAbsolute:= Tc3_HBI_System.cABORTED;
				END_IF
				IF FB_MC2_Compact_M_nMC_MoveAbsolute_fbMC2_MoveAbsolute2.Execute AND FB_MC2_Compact_M_nMC_MoveAbsolute_fbMC2_MoveAbsolute2.CommandAborted THEN
					M_nMC_MoveAbsolute:= Tc3_HBI_System.cABORTED;
				END_IF
			ELSE
				FB_MC2_Compact_M_nMC_MoveAbsolute_fbMC2_MoveAbsolute1(Axis:= _stAXIS_REF, Execute:= FALSE);
				FB_MC2_Compact_M_nMC_MoveAbsolute_fbMC2_MoveAbsolute2(Axis:= _stAXIS_REF, Execute:= FALSE);
				FB_MC2_Compact_M_nMC_MoveAbsolute_iState:= 000;
			END_IF
		
ELSE	
	FB_MC2_Compact_M_nMC_MoveAbsolute_iState:= 000;
END_CASE
END_METHOD

//	The result of the method is an unsigned double integer
//	0 = idle 
//	1 = coupled
//	2 = starting
//	3 = running
//	4 = aborted
// 	5 = no hardware connected
// 	6 = Spare
//	7 = pointer or index error
//	8 = mapping error
//	9 = parameter error
//	10 = complete
//	Any other number = ErrorID
METHOD PUBLIC M_nMC_MoveModulo : UDINT
VAR_INPUT
	bExecute: BOOL;
	lrPosition: LREAL;
	lrVelocity: LREAL;
	eDirection: Tc2_MC2.MC_Direction;
END_VAR
// Local variable
FB_MC2_Compact_M_nMC_MoveModulo_bExecute:= bExecute;
FB_MC2_Compact_M_nMC_MoveModulo_lrPosition:= lrPosition;
FB_MC2_Compact_M_nMC_MoveModulo_lrVelocity:= lrVelocity;
FB_MC2_Compact_M_nMC_MoveModulo_eDirection:= eDirection;

//**********************************
// Reset 
//**********************************
IF _bReset THEN
	IF _bError THEN
		FB_MC2_Compact_M_nMC_MoveModulo_fbMC2_MoveModulo1(Axis:= _stAXIS_REF, Execute:= FALSE);
		FB_MC2_Compact_M_nMC_MoveModulo_fbMC2_MoveModulo2(Axis:= _stAXIS_REF, Execute:= FALSE);
		FB_MC2_Compact_M_nMC_MoveModulo_iState:= 000;
		_sMessage:= '';
	END_IF		
END_IF

//**********************************
// Wait for execute
//**********************************
IF _stAXIS_REF.NcToPlc.AxisID > 0 THEN
	FB_MC2_Compact_M_nMC_MoveModulo_fbExecute_R_TRIG(CLK:= FB_MC2_Compact_M_nMC_MoveModulo_bExecute);
	IF FB_MC2_Compact_M_nMC_MoveModulo_fbExecute_R_TRIG.Q THEN
		FB_MC2_Compact_M_nMC_MoveModulo_fbMC2_MoveModulo1(Axis:= _stAXIS_REF, Position:= FB_MC2_Compact_M_nMC_MoveModulo_lrPosition, Velocity:= FB_MC2_Compact_M_nMC_MoveModulo_lrVelocity, Acceleration:= _stDynamic.lrAcceleration, Deceleration:= _stDynamic.lrDeceleration, Jerk:= _stDynamic.lrJerk, Direction:= FB_MC2_Compact_M_nMC_MoveModulo_eDirection, BufferMode:= _eBufferMode); 
		FB_MC2_Compact_M_nMC_MoveModulo_fbMC2_MoveModulo2(Axis:= _stAXIS_REF, Position:= FB_MC2_Compact_M_nMC_MoveModulo_lrPosition, Velocity:= FB_MC2_Compact_M_nMC_MoveModulo_lrVelocity, Acceleration:= _stDynamic.lrAcceleration, Deceleration:= _stDynamic.lrDeceleration, Jerk:= _stDynamic.lrJerk, Direction:= FB_MC2_Compact_M_nMC_MoveModulo_eDirection, BufferMode:= _eBufferMode); 
		
		// Axis not coupled	
		IF NOT _stAXIS_REF.Status.Coupled THEN
			IF FB_MC2_Compact_M_nMC_MoveModulo_fbMC2_MoveModulo1.Execute OR FB_MC2_Compact_M_nMC_MoveModulo_fbMC2_MoveModulo1.Busy THEN
				FB_MC2_Compact_M_nMC_MoveModulo_fbMC2_MoveModulo1(Axis:= _stAXIS_REF, Execute:= FALSE);
				FB_MC2_Compact_M_nMC_MoveModulo_fbMC2_MoveModulo2(Axis:= _stAXIS_REF, Execute:= FALSE);
				FB_MC2_Compact_M_nMC_MoveModulo_fbMC2_MoveModulo2.Execute:= TRUE;
				FB_MC2_Compact_M_nMC_MoveModulo_iState:= 010;
			ELSE	
				FB_MC2_Compact_M_nMC_MoveModulo_fbMC2_MoveModulo1(Axis:= _stAXIS_REF, Execute:= FALSE);
				FB_MC2_Compact_M_nMC_MoveModulo_fbMC2_MoveModulo2(Axis:= _stAXIS_REF, Execute:= FALSE);
				FB_MC2_Compact_M_nMC_MoveModulo_fbMC2_MoveModulo1.Execute:= TRUE;
				FB_MC2_Compact_M_nMC_MoveModulo_iState:= 001;
			END_IF	
		ELSE
			FB_MC2_Compact_M_nMC_MoveModulo_fbMC2_MoveModulo1(Axis:= _stAXIS_REF, Execute:= FALSE);
			FB_MC2_Compact_M_nMC_MoveModulo_fbMC2_MoveModulo2(Axis:= _stAXIS_REF, Execute:= FALSE);
			FB_MC2_Compact_M_nMC_MoveModulo_iState:= 030;
		END_IF
		
	END_IF
ELSE
	FB_MC2_Compact_M_nMC_MoveModulo_fbExecute_R_TRIG(CLK:= FALSE);
	FB_MC2_Compact_M_nMC_MoveModulo_iState:= 000;
	IF FB_MC2_Compact_M_nMC_MoveModulo_bExecute THEN
		M_nMC_MoveModulo:= Tc3_HBI_System.cMAPPING_ERROR;
	END_IF
	RETURN;
END_IF


//**********************************
// Main sequence
//**********************************
CASE FB_MC2_Compact_M_nMC_MoveModulo_iState OF

	000:	// Do nothing

	001:	// MoveModulo1 active
			M_nMC_MoveModulo:= Tc3_HBI_System.cSTARTING;
			FB_MC2_Compact_M_nMC_MoveModulo_fbMC2_MoveModulo1(Axis:= _stAXIS_REF);
			FB_MC2_Compact_M_nMC_MoveModulo_fbMC2_MoveModulo2(Axis:= _stAXIS_REF);
	
			// Command aborted
			IF FB_MC2_Compact_M_nMC_MoveModulo_fbMC2_MoveModulo1.CommandAborted THEN
				FB_MC2_Compact_M_nMC_MoveModulo_fbMC2_MoveModulo2.Execute:= FALSE; 
				FB_MC2_Compact_M_nMC_MoveModulo_iState:= 040;
			ELSE
				// Error handling
				IF FB_MC2_Compact_M_nMC_MoveModulo_fbMC2_MoveModulo1.Error THEN
					M_nError(nErrorID:= FB_MC2_Compact_M_nMC_MoveModulo_fbMC2_MoveModulo1.ErrorID);
					M_nMC_MoveModulo:= FB_MC2_Compact_M_nMC_MoveModulo_fbMC2_MoveModulo1.ErrorID;
					_sMessage:= 'Axis Move Modulo Error';
				ELSE
					// Active
					IF FB_MC2_Compact_M_nMC_MoveModulo_fbMC2_MoveModulo1.Active THEN
						FB_MC2_Compact_M_nMC_MoveModulo_iState:= 002;
					ELSE
						// Done
						IF FB_MC2_Compact_M_nMC_MoveModulo_fbMC2_MoveModulo1.Done THEN
							FB_MC2_Compact_M_nMC_MoveModulo_iState:= 040;
						END_IF
					END_IF	
				END_IF
			END_IF
			
	002:	// MoveModulo1 done
			M_nMC_MoveModulo:= Tc3_HBI_System.cRUNNING;
			FB_MC2_Compact_M_nMC_MoveModulo_fbMC2_MoveModulo1(Axis:= _stAXIS_REF);
			FB_MC2_Compact_M_nMC_MoveModulo_fbMC2_MoveModulo2(Axis:= _stAXIS_REF);
	
			// Command aborted
			IF FB_MC2_Compact_M_nMC_MoveModulo_fbMC2_MoveModulo1.CommandAborted THEN
				FB_MC2_Compact_M_nMC_MoveModulo_fbMC2_MoveModulo2.Execute:= FALSE; 
				FB_MC2_Compact_M_nMC_MoveModulo_iState:= 040;
			ELSE
				// Error handling
				IF FB_MC2_Compact_M_nMC_MoveModulo_fbMC2_MoveModulo1.Error THEN
					M_nError(nErrorID:= FB_MC2_Compact_M_nMC_MoveModulo_fbMC2_MoveModulo1.ErrorID);
					M_nMC_MoveModulo:= FB_MC2_Compact_M_nMC_MoveModulo_fbMC2_MoveModulo1.ErrorID;
					_sMessage:= 'Axis Move Modulo Error';
				ELSE
					// Done
					IF FB_MC2_Compact_M_nMC_MoveModulo_fbMC2_MoveModulo1.Done THEN
						FB_MC2_Compact_M_nMC_MoveModulo_iState:= 040;
					END_IF	
				END_IF
			END_IF

	010:	// Call MoveModulo2 active 
			M_nMC_MoveModulo:= Tc3_HBI_System.cSTARTING;
			FB_MC2_Compact_M_nMC_MoveModulo_fbMC2_MoveModulo1(Axis:= _stAXIS_REF);
			FB_MC2_Compact_M_nMC_MoveModulo_fbMC2_MoveModulo2(Axis:= _stAXIS_REF);
		
			// Command aborted
			IF FB_MC2_Compact_M_nMC_MoveModulo_fbMC2_MoveModulo2.CommandAborted THEN
				FB_MC2_Compact_M_nMC_MoveModulo_fbMC2_MoveModulo1.Execute:= FALSE; 
				FB_MC2_Compact_M_nMC_MoveModulo_iState:= 040;
			ELSE
				// Error handling
				IF FB_MC2_Compact_M_nMC_MoveModulo_fbMC2_MoveModulo2.Error THEN
					M_nError(nErrorID:= FB_MC2_Compact_M_nMC_MoveModulo_fbMC2_MoveModulo2.ErrorID);
					M_nMC_MoveModulo:= FB_MC2_Compact_M_nMC_MoveModulo_fbMC2_MoveModulo2.ErrorID;
					_sMessage:= 'Axis Move Modulo Error';
				ELSE
					// Active
					IF FB_MC2_Compact_M_nMC_MoveModulo_fbMC2_MoveModulo2.Active THEN
						FB_MC2_Compact_M_nMC_MoveModulo_iState:= 011;
					ELSE
						// Done
						IF FB_MC2_Compact_M_nMC_MoveModulo_fbMC2_MoveModulo2.Done THEN
							FB_MC2_Compact_M_nMC_MoveModulo_iState:= 040;
						END_IF
					END_IF	
				END_IF
			END_IF

	011:	// MoveModulo2 done
			M_nMC_MoveModulo:= Tc3_HBI_System.cRUNNING;
			FB_MC2_Compact_M_nMC_MoveModulo_fbMC2_MoveModulo1(Axis:= _stAXIS_REF);
			FB_MC2_Compact_M_nMC_MoveModulo_fbMC2_MoveModulo2(Axis:= _stAXIS_REF);
			
			// Command aborted
			IF FB_MC2_Compact_M_nMC_MoveModulo_fbMC2_MoveModulo2.CommandAborted THEN
				FB_MC2_Compact_M_nMC_MoveModulo_fbMC2_MoveModulo1.Execute:= FALSE; 
				FB_MC2_Compact_M_nMC_MoveModulo_iState:= 040;
			ELSE
				// Error handling
				IF FB_MC2_Compact_M_nMC_MoveModulo_fbMC2_MoveModulo2.Error THEN
					M_nError(nErrorID:= FB_MC2_Compact_M_nMC_MoveModulo_fbMC2_MoveModulo2.ErrorID);
					M_nMC_MoveModulo:= FB_MC2_Compact_M_nMC_MoveModulo_fbMC2_MoveModulo2.ErrorID;
					_sMessage:= 'Axis Move Modulo Error';
				ELSE
					// Done
					IF FB_MC2_Compact_M_nMC_MoveModulo_fbMC2_MoveModulo2.Done THEN
						FB_MC2_Compact_M_nMC_MoveModulo_iState:= 040;
					END_IF	
				END_IF	
			END_IF

	030: // Coupled
			M_nMC_MoveModulo:= Tc3_HBI_System.cCOUPLED;
			FB_MC2_Compact_M_nMC_MoveModulo_fbMC2_MoveModulo1(Axis:= _stAXIS_REF);
			FB_MC2_Compact_M_nMC_MoveModulo_fbMC2_MoveModulo2(Axis:= _stAXIS_REF);

			IF NOT FB_MC2_Compact_M_nMC_MoveModulo_bExecute THEN
				FB_MC2_Compact_M_nMC_MoveModulo_fbMC2_MoveModulo1(Axis:= _stAXIS_REF, Execute:= FALSE);
				FB_MC2_Compact_M_nMC_MoveModulo_fbMC2_MoveModulo2(Axis:= _stAXIS_REF, Execute:= FALSE);
				FB_MC2_Compact_M_nMC_MoveModulo_iState:= 000;
			END_IF

	040:	// Done
			M_nMC_MoveModulo:= Tc3_HBI_System.cCOMPLETE;
			FB_MC2_Compact_M_nMC_MoveModulo_fbMC2_MoveModulo1(Axis:= _stAXIS_REF);
			FB_MC2_Compact_M_nMC_MoveModulo_fbMC2_MoveModulo2(Axis:= _stAXIS_REF);

			IF FB_MC2_Compact_M_nMC_MoveModulo_bExecute THEN			
				IF FB_MC2_Compact_M_nMC_MoveModulo_fbMC2_MoveModulo1.Execute AND FB_MC2_Compact_M_nMC_MoveModulo_fbMC2_MoveModulo1.CommandAborted THEN
					M_nMC_MoveModulo:= Tc3_HBI_System.cABORTED;
				END_IF
				IF FB_MC2_Compact_M_nMC_MoveModulo_fbMC2_MoveModulo2.Execute AND FB_MC2_Compact_M_nMC_MoveModulo_fbMC2_MoveModulo2.CommandAborted THEN
					M_nMC_MoveModulo:= Tc3_HBI_System.cABORTED;
				END_IF
			ELSE	
				FB_MC2_Compact_M_nMC_MoveModulo_fbMC2_MoveModulo1(Axis:= _stAXIS_REF, Execute:= FALSE);
				FB_MC2_Compact_M_nMC_MoveModulo_fbMC2_MoveModulo2(Axis:= _stAXIS_REF, Execute:= FALSE);
				FB_MC2_Compact_M_nMC_MoveModulo_iState:= 000;
			END_IF
		
ELSE	
	FB_MC2_Compact_M_nMC_MoveModulo_iState:= 000;
END_CASE
END_METHOD

//	The result of the method is an unsigned double integer
//	0 = idle 
//	1 = coupled
//	2 = starting
//	3 = running
//	4 = aborted
// 	5 = no hardware connected
// 	6 = Spare
//	7 = pointer or index error
//	8 = mapping error
//	9 = parameter error
//	10 = complete
//	Any other number = ErrorID
METHOD PUBLIC M_nMC_MoveRelative : UDINT
VAR_INPUT
	bExecute: BOOL;
	lrDistance: LREAL;
	lrVelocity: LREAL;
END_VAR
// Local variable
FB_MC2_Compact_M_nMC_MoveRelative_bExecute:= bExecute;
FB_MC2_Compact_M_nMC_MoveRelative_lrDistance:= lrDistance;
FB_MC2_Compact_M_nMC_MoveRelative_lrVelocity:= lrVelocity;

//**********************************
// Reset 
//**********************************
IF _bReset THEN
	IF _bError THEN
		FB_MC2_Compact_M_nMC_MoveRelative_fbMC2_MoveRelative1(Axis:= _stAXIS_REF, Execute:= FALSE);
		FB_MC2_Compact_M_nMC_MoveRelative_fbMC2_MoveRelative2(Axis:= _stAXIS_REF, Execute:= FALSE);
		FB_MC2_Compact_M_nMC_MoveRelative_iState:= 000;
		_sMessage:= '';
	END_IF		
END_IF

//**********************************
// Wait for execute
//**********************************
IF _stAXIS_REF.NcToPlc.AxisID > 0 THEN
	FB_MC2_Compact_M_nMC_MoveRelative_fbExecute_R_TRIG(CLK:= FB_MC2_Compact_M_nMC_MoveRelative_bExecute);
	IF FB_MC2_Compact_M_nMC_MoveRelative_fbExecute_R_TRIG.Q THEN
		FB_MC2_Compact_M_nMC_MoveRelative_fbMC2_MoveRelative1(Axis:= _stAXIS_REF, Distance:= FB_MC2_Compact_M_nMC_MoveRelative_lrDistance, Velocity:= FB_MC2_Compact_M_nMC_MoveRelative_lrVelocity, Acceleration:= _stDynamic.lrAcceleration, Deceleration:= _stDynamic.lrDeceleration, Jerk:= _stDynamic.lrJerk, BufferMode:= _eBufferMode); 
		FB_MC2_Compact_M_nMC_MoveRelative_fbMC2_MoveRelative2(Axis:= _stAXIS_REF, Distance:= FB_MC2_Compact_M_nMC_MoveRelative_lrDistance, Velocity:= FB_MC2_Compact_M_nMC_MoveRelative_lrVelocity, Acceleration:= _stDynamic.lrAcceleration, Deceleration:= _stDynamic.lrDeceleration, Jerk:= _stDynamic.lrJerk, BufferMode:= _eBufferMode); 
	
		// Axis not coupled	
		IF NOT _stAXIS_REF.Status.Coupled THEN
			IF FB_MC2_Compact_M_nMC_MoveRelative_fbMC2_MoveRelative1.Execute OR FB_MC2_Compact_M_nMC_MoveRelative_fbMC2_MoveRelative1.Busy THEN
				FB_MC2_Compact_M_nMC_MoveRelative_fbMC2_MoveRelative1(Axis:= _stAXIS_REF, Execute:= FALSE);
				FB_MC2_Compact_M_nMC_MoveRelative_fbMC2_MoveRelative2(Axis:= _stAXIS_REF, Execute:= FALSE);
				FB_MC2_Compact_M_nMC_MoveRelative_fbMC2_MoveRelative2.Execute:= TRUE;
				FB_MC2_Compact_M_nMC_MoveRelative_iState:= 010;
			ELSE
				FB_MC2_Compact_M_nMC_MoveRelative_fbMC2_MoveRelative1(Axis:= _stAXIS_REF, Execute:= FALSE);
				FB_MC2_Compact_M_nMC_MoveRelative_fbMC2_MoveRelative2(Axis:= _stAXIS_REF, Execute:= FALSE);
				FB_MC2_Compact_M_nMC_MoveRelative_fbMC2_MoveRelative1.Execute:= TRUE;
				FB_MC2_Compact_M_nMC_MoveRelative_iState:= 001;
			END_IF
		ELSE
			FB_MC2_Compact_M_nMC_MoveRelative_fbMC2_MoveRelative1(Axis:= _stAXIS_REF, Execute:= FALSE);
			FB_MC2_Compact_M_nMC_MoveRelative_fbMC2_MoveRelative2(Axis:= _stAXIS_REF, Execute:= FALSE);
			FB_MC2_Compact_M_nMC_MoveRelative_iState:= 030;
		END_IF
	
	END_IF
ELSE
	FB_MC2_Compact_M_nMC_MoveRelative_fbExecute_R_TRIG(CLK:= FALSE);
	FB_MC2_Compact_M_nMC_MoveRelative_iState:= 000;
	IF FB_MC2_Compact_M_nMC_MoveRelative_bExecute THEN
		M_nMC_MoveRelative:= Tc3_HBI_System.cMAPPING_ERROR;
	END_IF
	RETURN;
END_IF


//**********************************
// Main sequence
//**********************************
CASE FB_MC2_Compact_M_nMC_MoveRelative_iState OF

	000:	// Do nothing

	001:	// Call MoveRelative1 active 
			M_nMC_MoveRelative:= Tc3_HBI_System.cSTARTING;
			FB_MC2_Compact_M_nMC_MoveRelative_fbMC2_MoveRelative1(Axis:= _stAXIS_REF); 
			FB_MC2_Compact_M_nMC_MoveRelative_fbMC2_MoveRelative2(Axis:= _stAXIS_REF); 
	
			// Command aborted
			IF FB_MC2_Compact_M_nMC_MoveRelative_fbMC2_MoveRelative1.CommandAborted THEN
				FB_MC2_Compact_M_nMC_MoveRelative_fbMC2_MoveRelative2.Execute:= FALSE; 
				FB_MC2_Compact_M_nMC_MoveRelative_iState:= 040;
			ELSE
				// Error handling
				IF FB_MC2_Compact_M_nMC_MoveRelative_fbMC2_MoveRelative1.Error THEN
					M_nError(nErrorID:= FB_MC2_Compact_M_nMC_MoveRelative_fbMC2_MoveRelative1.ErrorID);
					M_nMC_MoveRelative:= FB_MC2_Compact_M_nMC_MoveRelative_fbMC2_MoveRelative1.ErrorID;
					_sMessage:= 'Axis Move Relative Error';
				ELSE
					// Active
					IF FB_MC2_Compact_M_nMC_MoveRelative_fbMC2_MoveRelative1.Active THEN
						FB_MC2_Compact_M_nMC_MoveRelative_iState:= 002;
					ELSE
						// Done
						IF FB_MC2_Compact_M_nMC_MoveRelative_fbMC2_MoveRelative1.Done THEN
							FB_MC2_Compact_M_nMC_MoveRelative_iState:= 040;
						END_IF
					END_IF	
				END_IF
			END_IF
			
	002:	// MoveRelative1 done
			M_nMC_MoveRelative:= Tc3_HBI_System.cRUNNING;
			FB_MC2_Compact_M_nMC_MoveRelative_fbMC2_MoveRelative1(Axis:= _stAXIS_REF); 
			FB_MC2_Compact_M_nMC_MoveRelative_fbMC2_MoveRelative2(Axis:= _stAXIS_REF); 
	
			// Command aborted
			IF FB_MC2_Compact_M_nMC_MoveRelative_fbMC2_MoveRelative1.CommandAborted THEN
				FB_MC2_Compact_M_nMC_MoveRelative_fbMC2_MoveRelative2.Execute:= FALSE; 
				FB_MC2_Compact_M_nMC_MoveRelative_iState:= 040;
			ELSE
				// Error handling
				IF FB_MC2_Compact_M_nMC_MoveRelative_fbMC2_MoveRelative1.Error THEN
					M_nError(nErrorID:= FB_MC2_Compact_M_nMC_MoveRelative_fbMC2_MoveRelative1.ErrorID);
					M_nMC_MoveRelative:= FB_MC2_Compact_M_nMC_MoveRelative_fbMC2_MoveRelative1.ErrorID;
					_sMessage:= 'Axis Move Relative Error';
				ELSE
					// Done
					IF FB_MC2_Compact_M_nMC_MoveRelative_fbMC2_MoveRelative1.Done THEN
						FB_MC2_Compact_M_nMC_MoveRelative_iState:= 040;
					END_IF	
				END_IF
			END_IF

	010:	// MoveRelative2 active 
			M_nMC_MoveRelative:= Tc3_HBI_System.cSTARTING;
			FB_MC2_Compact_M_nMC_MoveRelative_fbMC2_MoveRelative1(Axis:= _stAXIS_REF); 
			FB_MC2_Compact_M_nMC_MoveRelative_fbMC2_MoveRelative2(Axis:= _stAXIS_REF); 
			
			// Command aborted
			IF FB_MC2_Compact_M_nMC_MoveRelative_fbMC2_MoveRelative2.CommandAborted THEN
				FB_MC2_Compact_M_nMC_MoveRelative_fbMC2_MoveRelative1.Execute:= FALSE; 
				FB_MC2_Compact_M_nMC_MoveRelative_iState:= 040;
			ELSE
				// Error handling
				IF FB_MC2_Compact_M_nMC_MoveRelative_fbMC2_MoveRelative2.Error THEN
					M_nError(nErrorID:= FB_MC2_Compact_M_nMC_MoveRelative_fbMC2_MoveRelative2.ErrorID);
					M_nMC_MoveRelative:= FB_MC2_Compact_M_nMC_MoveRelative_fbMC2_MoveRelative2.ErrorID;
					_sMessage:= 'Axis Move Relative Error';
				ELSE
					// Active
					IF FB_MC2_Compact_M_nMC_MoveRelative_fbMC2_MoveRelative2.Active THEN
						FB_MC2_Compact_M_nMC_MoveRelative_iState:= 011;
					ELSE
						// Done
						IF FB_MC2_Compact_M_nMC_MoveRelative_fbMC2_MoveRelative2.Done THEN
							FB_MC2_Compact_M_nMC_MoveRelative_iState:= 040;
						END_IF
					END_IF	
				END_IF
			END_IF
		
	011:	// MoveRelative2 done
			M_nMC_MoveRelative:= Tc3_HBI_System.cRUNNING;
			FB_MC2_Compact_M_nMC_MoveRelative_fbMC2_MoveRelative1(Axis:= _stAXIS_REF); 
			FB_MC2_Compact_M_nMC_MoveRelative_fbMC2_MoveRelative2(Axis:= _stAXIS_REF); 
			
			// Command aborted
			IF FB_MC2_Compact_M_nMC_MoveRelative_fbMC2_MoveRelative2.CommandAborted THEN
				FB_MC2_Compact_M_nMC_MoveRelative_fbMC2_MoveRelative1.Execute:= FALSE; 
				FB_MC2_Compact_M_nMC_MoveRelative_iState:= 040;
			ELSE
				// Error handling
				IF FB_MC2_Compact_M_nMC_MoveRelative_fbMC2_MoveRelative2.Error THEN
					M_nError(nErrorID:= FB_MC2_Compact_M_nMC_MoveRelative_fbMC2_MoveRelative2.ErrorID);
					M_nMC_MoveRelative:= FB_MC2_Compact_M_nMC_MoveRelative_fbMC2_MoveRelative2.ErrorID;
					_sMessage:= 'Axis Move Relative Error';
				ELSE
					// Done
					IF FB_MC2_Compact_M_nMC_MoveRelative_fbMC2_MoveRelative2.Done THEN
						FB_MC2_Compact_M_nMC_MoveRelative_iState:= 040;
					END_IF	
				END_IF	
			END_IF
	
	030: // Coupled
			M_nMC_MoveRelative:= Tc3_HBI_System.cCOUPLED;
			FB_MC2_Compact_M_nMC_MoveRelative_fbMC2_MoveRelative1(Axis:= _stAXIS_REF); 
			FB_MC2_Compact_M_nMC_MoveRelative_fbMC2_MoveRelative2(Axis:= _stAXIS_REF); 

			IF NOT FB_MC2_Compact_M_nMC_MoveRelative_bExecute THEN
				FB_MC2_Compact_M_nMC_MoveRelative_fbMC2_MoveRelative1(Axis:= _stAXIS_REF, Execute:= FALSE);
				FB_MC2_Compact_M_nMC_MoveRelative_fbMC2_MoveRelative2(Axis:= _stAXIS_REF, Execute:= FALSE);
				FB_MC2_Compact_M_nMC_MoveRelative_iState:= 000;
			END_IF

	040: // Done
			M_nMC_MoveRelative:= Tc3_HBI_System.cCOMPLETE;
			FB_MC2_Compact_M_nMC_MoveRelative_fbMC2_MoveRelative1(Axis:= _stAXIS_REF); 
			FB_MC2_Compact_M_nMC_MoveRelative_fbMC2_MoveRelative2(Axis:= _stAXIS_REF); 

			IF FB_MC2_Compact_M_nMC_MoveRelative_bExecute THEN			
				IF FB_MC2_Compact_M_nMC_MoveRelative_fbMC2_MoveRelative1.Execute AND FB_MC2_Compact_M_nMC_MoveRelative_fbMC2_MoveRelative1.CommandAborted THEN
					M_nMC_MoveRelative:= Tc3_HBI_System.cABORTED;
				END_IF
				IF FB_MC2_Compact_M_nMC_MoveRelative_fbMC2_MoveRelative2.Execute AND FB_MC2_Compact_M_nMC_MoveRelative_fbMC2_MoveRelative2.CommandAborted THEN
					M_nMC_MoveRelative:= Tc3_HBI_System.cABORTED;
				END_IF
			ELSE
				FB_MC2_Compact_M_nMC_MoveRelative_fbMC2_MoveRelative1(Axis:= _stAXIS_REF, Execute:= FALSE);
				FB_MC2_Compact_M_nMC_MoveRelative_fbMC2_MoveRelative2(Axis:= _stAXIS_REF, Execute:= FALSE);
				FB_MC2_Compact_M_nMC_MoveRelative_iState:= 000;
			END_IF
		
ELSE	
	FB_MC2_Compact_M_nMC_MoveRelative_iState:= 000;
END_CASE
END_METHOD

//	The result of the method is an unsigned double integer
//	0 = idle 
//	1 = coupled
//	2 = starting
//	3 = running
//	4 = aborted
// 	5 = no hardware connected
// 	6 = Spare
//	7 = pointer or index error
//	8 = mapping error
//	9 = parameter error
//	10 = complete
//	Any other number = ErrorID
METHOD PUBLIC M_nMC_MoveVelocity : UDINT
VAR_INPUT
	bExecute: BOOL;
	lrVelocity: LREAL;
	eDirection: MC_Direction;
END_VAR
// Local variable
FB_MC2_Compact_M_nMC_MoveVelocity_bExecute:= bExecute;
FB_MC2_Compact_M_nMC_MoveVelocity_lrVelocity:= lrVelocity;
FB_MC2_Compact_M_nMC_MoveVelocity_eDirection:= eDirection;

//**********************************
// Reset 
//**********************************
IF _bReset THEN
	IF _bError THEN	
		FB_MC2_Compact_M_nMC_MoveVelocity_fbMC2_MoveVelocity1(Axis:= _stAXIS_REF, Execute:= FALSE);
		FB_MC2_Compact_M_nMC_MoveVelocity_fbMC2_MoveVelocity2(Axis:= _stAXIS_REF, Execute:= FALSE);
		FB_MC2_Compact_M_nMC_MoveVelocity_iState:= 000;
		_sMessage:= '';
	END_IF
END_IF

//**********************************
// Wait for execute
//**********************************
IF _stAXIS_REF.NcToPlc.AxisID > 0 THEN
	FB_MC2_Compact_M_nMC_MoveVelocity_fbExecute_R_TRIG(CLK:= FB_MC2_Compact_M_nMC_MoveVelocity_bExecute);
	IF FB_MC2_Compact_M_nMC_MoveVelocity_fbExecute_R_TRIG.Q THEN
		FB_MC2_Compact_M_nMC_MoveVelocity_fbMC2_MoveVelocity1(Axis:= _stAXIS_REF, Velocity:= FB_MC2_Compact_M_nMC_MoveVelocity_lrVelocity, Acceleration:= _stDynamic.lrAcceleration, Deceleration:= _stDynamic.lrDeceleration, Jerk:= _stDynamic.lrJerk, Direction:= FB_MC2_Compact_M_nMC_MoveVelocity_eDirection, BufferMode:= _eBufferMode); 
		FB_MC2_Compact_M_nMC_MoveVelocity_fbMC2_MoveVelocity2(Axis:= _stAXIS_REF, Velocity:= FB_MC2_Compact_M_nMC_MoveVelocity_lrVelocity, Acceleration:= _stDynamic.lrAcceleration, Deceleration:= _stDynamic.lrDeceleration, Jerk:= _stDynamic.lrJerk, Direction:= FB_MC2_Compact_M_nMC_MoveVelocity_eDirection, BufferMode:= _eBufferMode); 
		
		// Axis not coupled	
		IF NOT _stAXIS_REF.Status.Coupled THEN
			IF FB_MC2_Compact_M_nMC_MoveVelocity_fbMC2_MoveVelocity1.Active OR FB_MC2_Compact_M_nMC_MoveVelocity_fbMC2_MoveVelocity1.Busy THEN
				FB_MC2_Compact_M_nMC_MoveVelocity_fbMC2_MoveVelocity1(Axis:= _stAXIS_REF, Execute:= FALSE);
				FB_MC2_Compact_M_nMC_MoveVelocity_fbMC2_MoveVelocity2(Axis:= _stAXIS_REF, Execute:= FALSE);
				FB_MC2_Compact_M_nMC_MoveVelocity_fbMC2_MoveVelocity2.Execute:= TRUE; 
				FB_MC2_Compact_M_nMC_MoveVelocity_iState:= 010;
			ELSE
				FB_MC2_Compact_M_nMC_MoveVelocity_fbMC2_MoveVelocity1(Axis:= _stAXIS_REF, Execute:= FALSE);
				FB_MC2_Compact_M_nMC_MoveVelocity_fbMC2_MoveVelocity2(Axis:= _stAXIS_REF, Execute:= FALSE);
				FB_MC2_Compact_M_nMC_MoveVelocity_fbMC2_MoveVelocity1.Execute:= TRUE; 
				FB_MC2_Compact_M_nMC_MoveVelocity_iState:= 001;
			END_IF
		ELSE
			FB_MC2_Compact_M_nMC_MoveVelocity_fbMC2_MoveVelocity1(Axis:= _stAXIS_REF, Execute:= FALSE);
			FB_MC2_Compact_M_nMC_MoveVelocity_fbMC2_MoveVelocity2(Axis:= _stAXIS_REF, Execute:= FALSE);
			FB_MC2_Compact_M_nMC_MoveVelocity_iState:= 030;
		END_IF
		
	END_IF
ELSE
	FB_MC2_Compact_M_nMC_MoveVelocity_fbExecute_R_TRIG(CLK:= FALSE);
	FB_MC2_Compact_M_nMC_MoveVelocity_iState:= 000;
	IF FB_MC2_Compact_M_nMC_MoveVelocity_bExecute THEN
		M_nMC_MoveVelocity:= Tc3_HBI_System.cMAPPING_ERROR;
	END_IF
	RETURN;
END_IF


//**********************************
// Main sequence
//**********************************
CASE FB_MC2_Compact_M_nMC_MoveVelocity_iState OF

	000:	// Do nothing

	001:	// MoveVelocity1 active
			M_nMC_MoveVelocity:= Tc3_HBI_System.cSTARTING;
			FB_MC2_Compact_M_nMC_MoveVelocity_fbMC2_MoveVelocity1(Axis:= _stAXIS_REF);
			FB_MC2_Compact_M_nMC_MoveVelocity_fbMC2_MoveVelocity2(Axis:= _stAXIS_REF);
				
			// Command aborted
			IF FB_MC2_Compact_M_nMC_MoveVelocity_fbMC2_MoveVelocity1.CommandAborted THEN
				FB_MC2_Compact_M_nMC_MoveVelocity_fbMC2_MoveVelocity2.Execute:= FALSE; 
				FB_MC2_Compact_M_nMC_MoveVelocity_iState:= 040;
			ELSE
				// Error handling
				IF FB_MC2_Compact_M_nMC_MoveVelocity_fbMC2_MoveVelocity1.Error THEN
					M_nError(nErrorID:= FB_MC2_Compact_M_nMC_MoveVelocity_fbMC2_MoveVelocity1.ErrorID);
					M_nMC_MoveVelocity:= FB_MC2_Compact_M_nMC_MoveVelocity_fbMC2_MoveVelocity1.ErrorID;
					_sMessage:= 'Axis Move Velocity Error';
				ELSE
					// Active
					IF FB_MC2_Compact_M_nMC_MoveVelocity_fbMC2_MoveVelocity1.Active THEN
						FB_MC2_Compact_M_nMC_MoveVelocity_iState:= 002;
					END_IF
				END_IF
			END_IF
	
	002:	// MoveVelocity1 done
			M_nMC_MoveVelocity:= Tc3_HBI_System.cRUNNING;
			FB_MC2_Compact_M_nMC_MoveVelocity_fbMC2_MoveVelocity1(Axis:= _stAXIS_REF);
			FB_MC2_Compact_M_nMC_MoveVelocity_fbMC2_MoveVelocity2(Axis:= _stAXIS_REF);
	
			// Command aborted
			IF FB_MC2_Compact_M_nMC_MoveVelocity_fbMC2_MoveVelocity1.CommandAborted THEN
				FB_MC2_Compact_M_nMC_MoveVelocity_fbMC2_MoveVelocity2.Execute:= FALSE; 
				FB_MC2_Compact_M_nMC_MoveVelocity_iState:= 040;
			ELSE
				// Error handling
				IF FB_MC2_Compact_M_nMC_MoveVelocity_fbMC2_MoveVelocity1.Error THEN
					M_nError(nErrorID:= FB_MC2_Compact_M_nMC_MoveVelocity_fbMC2_MoveVelocity1.ErrorID);
					M_nMC_MoveVelocity:= FB_MC2_Compact_M_nMC_MoveVelocity_fbMC2_MoveVelocity1.ErrorID;
					_sMessage:= 'Axis Move Velocity Error';
				ELSE
					// Done
					IF _stAXIS_REF.Status.ConstantVelocity THEN
						FB_MC2_Compact_M_nMC_MoveVelocity_iState:= 040;
					END_IF	
				END_IF
			END_IF
		
	010:	// MoveVelocity2 active 
			M_nMC_MoveVelocity:= Tc3_HBI_System.cSTARTING;
			FB_MC2_Compact_M_nMC_MoveVelocity_fbMC2_MoveVelocity1(Axis:= _stAXIS_REF);
			FB_MC2_Compact_M_nMC_MoveVelocity_fbMC2_MoveVelocity2(Axis:= _stAXIS_REF);
	
			// Command aborted
			IF FB_MC2_Compact_M_nMC_MoveVelocity_fbMC2_MoveVelocity2.CommandAborted THEN
				FB_MC2_Compact_M_nMC_MoveVelocity_fbMC2_MoveVelocity1.Execute:= FALSE; 
				FB_MC2_Compact_M_nMC_MoveVelocity_iState:= 040;
			ELSE
				// Error handling
				IF FB_MC2_Compact_M_nMC_MoveVelocity_fbMC2_MoveVelocity2.Error THEN
					M_nError(nErrorID:= FB_MC2_Compact_M_nMC_MoveVelocity_fbMC2_MoveVelocity2.ErrorID);
					M_nMC_MoveVelocity:= FB_MC2_Compact_M_nMC_MoveVelocity_fbMC2_MoveVelocity2.ErrorID;
					_sMessage:= 'Axis Move Velocity Error';
				ELSE
					// Active
					IF FB_MC2_Compact_M_nMC_MoveVelocity_fbMC2_MoveVelocity2.Active THEN
						FB_MC2_Compact_M_nMC_MoveVelocity_iState:= 011;
					END_IF	
				END_IF
			END_IF

	011:	// MoveVelocity2 done
			M_nMC_MoveVelocity:= Tc3_HBI_System.cRUNNING;
			FB_MC2_Compact_M_nMC_MoveVelocity_fbMC2_MoveVelocity1(Axis:= _stAXIS_REF);
			FB_MC2_Compact_M_nMC_MoveVelocity_fbMC2_MoveVelocity2(Axis:= _stAXIS_REF);
			
			// Command aborted
			IF FB_MC2_Compact_M_nMC_MoveVelocity_fbMC2_MoveVelocity2.CommandAborted THEN
				FB_MC2_Compact_M_nMC_MoveVelocity_fbMC2_MoveVelocity1.Execute:= FALSE; 
				FB_MC2_Compact_M_nMC_MoveVelocity_iState:= 040;
			ELSE
				// Error handling
				IF FB_MC2_Compact_M_nMC_MoveVelocity_fbMC2_MoveVelocity2.Error THEN
					M_nError(nErrorID:= FB_MC2_Compact_M_nMC_MoveVelocity_fbMC2_MoveVelocity2.ErrorID);
					M_nMC_MoveVelocity:= FB_MC2_Compact_M_nMC_MoveVelocity_fbMC2_MoveVelocity2.ErrorID;
					_sMessage:= 'Axis Move Velocity Error';
				ELSE
					// Done
					IF _stAXIS_REF.Status.ConstantVelocity THEN
						FB_MC2_Compact_M_nMC_MoveVelocity_iState:= 040;
					END_IF	
				END_IF	
			END_IF
			
	030: // Coupled
			M_nMC_MoveVelocity:= Tc3_HBI_System.cCOUPLED;
			FB_MC2_Compact_M_nMC_MoveVelocity_fbMC2_MoveVelocity1(Axis:= _stAXIS_REF);
			FB_MC2_Compact_M_nMC_MoveVelocity_fbMC2_MoveVelocity2(Axis:= _stAXIS_REF);

			IF NOT FB_MC2_Compact_M_nMC_MoveVelocity_bExecute THEN
				FB_MC2_Compact_M_nMC_MoveVelocity_fbMC2_MoveVelocity1(Axis:= _stAXIS_REF, Execute:= FALSE);
				FB_MC2_Compact_M_nMC_MoveVelocity_fbMC2_MoveVelocity2(Axis:= _stAXIS_REF, Execute:= FALSE);
				FB_MC2_Compact_M_nMC_MoveVelocity_iState:= 000;
			END_IF

	040: // Done
			M_nMC_MoveVelocity:= Tc3_HBI_System.cCOMPLETE;
			FB_MC2_Compact_M_nMC_MoveVelocity_fbMC2_MoveVelocity1(Axis:= _stAXIS_REF);
			FB_MC2_Compact_M_nMC_MoveVelocity_fbMC2_MoveVelocity2(Axis:= _stAXIS_REF);

			IF FB_MC2_Compact_M_nMC_MoveVelocity_bExecute THEN
				IF FB_MC2_Compact_M_nMC_MoveVelocity_fbMC2_MoveVelocity1.Execute AND FB_MC2_Compact_M_nMC_MoveVelocity_fbMC2_MoveVelocity1.CommandAborted THEN
					M_nMC_MoveVelocity:= Tc3_HBI_System.cABORTED;
				END_IF
				IF FB_MC2_Compact_M_nMC_MoveVelocity_fbMC2_MoveVelocity2.Execute AND FB_MC2_Compact_M_nMC_MoveVelocity_fbMC2_MoveVelocity2.CommandAborted THEN
					M_nMC_MoveVelocity:= Tc3_HBI_System.cABORTED;
				END_IF
			ELSE	
				FB_MC2_Compact_M_nMC_MoveVelocity_fbMC2_MoveVelocity1(Axis:= _stAXIS_REF, Execute:= FALSE);
				FB_MC2_Compact_M_nMC_MoveVelocity_fbMC2_MoveVelocity2(Axis:= _stAXIS_REF, Execute:= FALSE);
				FB_MC2_Compact_M_nMC_MoveVelocity_iState:= 000;
			END_IF
		
ELSE	
	FB_MC2_Compact_M_nMC_MoveVelocity_iState:= 000;
END_CASE
END_METHOD

//	The result of the method is an unsigned double integer
//	0 = idle 
//	1 = coupled
//	2 = starting
//	3 = running
//	4 = aborted
// 	5 = no hardware connected
// 	6 = Spare
//	7 = pointer or index error
//	8 = mapping error
//	9 = parameter error
//	10 = complete
//	Any other number = ErrorID
METHOD PUBLIC M_nMC_Power : UDINT
VAR_INPUT
	bEnable: BOOL;
	bE_Stop: BOOL;
	bE_StopDelay: BOOL;
	bEnable_Positive: BOOL;
	bEnable_Negative: BOOL;
END_VAR
// Update axis status
_stAXIS_REF.ReadStatus();

// Local variable
FB_MC2_Compact_M_nMC_Power_bEnable:= bEnable;
FB_MC2_Compact_M_nMC_Power_bE_Stop:= bE_Stop;
FB_MC2_Compact_M_nMC_Power_bE_StopDelay:= bE_StopDelay;
FB_MC2_Compact_M_nMC_Power_bEnable_Positive:= bEnable_Positive;
FB_MC2_Compact_M_nMC_Power_bEnable_Negative:= bEnable_Negative;

// Hardware conneted
_bHardwareConnected:= NOT BIT_TO_BOOL(_stAXIS_REF.NcToPlc.StateDWord.30) AND _stDriveAddress.SlaveAddress > 0 AND _stAXIS_REF.NcToPlc.AxisID > 0;

//**********************************
// Reset 
//**********************************
IF THIS^._bReset THEN
	MEMSET(destAddr:= ADR(FB_MC2_Compact_M_nMC_Power_arr_nRet), fillByte:= 16#00, n:= SIZEOF(FB_MC2_Compact_M_nMC_Power_arr_nRet));

	// Reset all methods
	M_nMC_Halt(bExecute:= FB_MC2_Compact_M_nMC_Halt_bExecute);
	M_nMC_Home(bExecute:= FB_MC2_Compact_M_nMC_Home_bExecute, lrPosition:= FB_MC2_Compact_M_nMC_Home_lrPosition, bCalibrationCam:= FB_MC2_Compact_M_nMC_Home_bCalibrationCam, eHomingMode:= FB_MC2_Compact_M_nMC_Home_eHomingMode);
	M_nMC_HomeReset(bExecute:= FB_MC2_Compact_M_nMC_HomeReset_bExecute);
	M_nMC_Jog(bForward:= FB_MC2_Compact_M_nMC_Jog_bForward, bBackwards:= FB_MC2_Compact_M_nMC_Jog_bBackwards, lrVelocity:= FB_MC2_Compact_M_nMC_Jog_lrVelocity);
	M_nMC_Local_Halt(bExecute:= FB_MC2_Compact_M_nMC_Local_Halt_bExecute);
	M_nMC_MoveAbsolute(bExecute:= FB_MC2_Compact_M_nMC_MoveAbsolute_bExecute, lrPosition:= FB_MC2_Compact_M_nMC_MoveAbsolute_lrPosition, lrVelocity:= FB_MC2_Compact_M_nMC_MoveAbsolute_lrVelocity);
	M_nMC_MoveModulo(bExecute:= FB_MC2_Compact_M_nMC_MoveModulo_bExecute, lrPosition:= FB_MC2_Compact_M_nMC_MoveModulo_lrPosition, lrVelocity:= FB_MC2_Compact_M_nMC_MoveModulo_lrVelocity, eDirection:= FB_MC2_Compact_M_nMC_MoveModulo_eDirection);
	M_nMC_MoveRelative(bExecute:= FB_MC2_Compact_M_nMC_MoveRelative_bExecute, lrDistance:= FB_MC2_Compact_M_nMC_MoveRelative_lrDistance, lrVelocity:= FB_MC2_Compact_M_nMC_MoveRelative_lrVelocity);
	M_nMC_MoveVelocity(bExecute:= FB_MC2_Compact_M_nMC_MoveVelocity_bExecute, lrVelocity:= FB_MC2_Compact_M_nMC_MoveVelocity_lrVelocity, eDirection:= FB_MC2_Compact_M_nMC_MoveVelocity_eDirection);
	M_nMC_QuickStop(bExecute:= FB_MC2_Compact_M_nMC_QuickStop_bExecute, lrDeceleration:= FB_MC2_Compact_M_nMC_QuickStop_lrDeceleration, lrJerk:= FB_MC2_Compact_M_nMC_QuickStop_lrJerk);
	M_nMC_ReadDriveAddress(bExecute:= FB_MC2_Compact_M_nMC_ReadDriveAddress_bExecute);
	M_nMC_Stop(bExecute:= FB_MC2_Compact_M_nMC_Stop_bExecute);
	_sMessage:= '';
END_IF

//***************************************
// Power 
//***************************************

